Yaskawa INFORM job: A_ROOF_UPPER_0614_2_PAINT_7.JBI

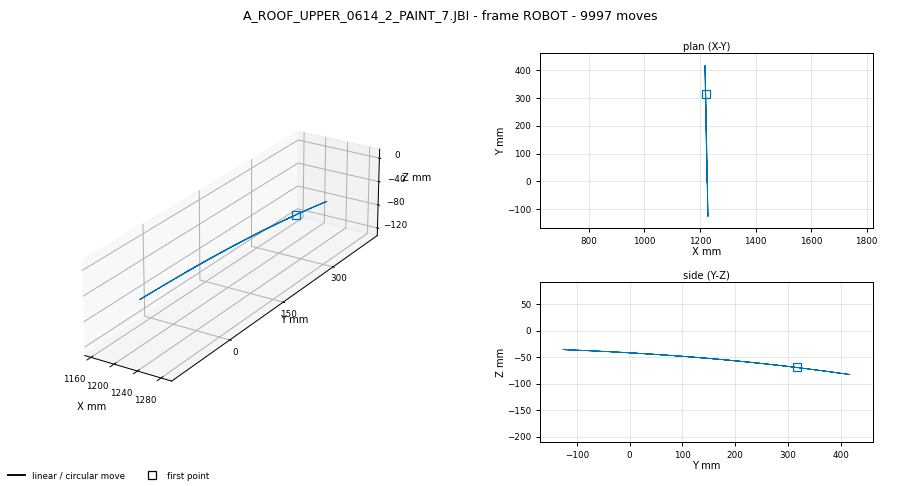
[picture p0: tool path of A_ROOF_UPPER_0614_2_PAINT_7.JBI in frame ROBOT, 9997 of 9997 moves have a stored position in this frame; points joined in program order, loops and branches not executed]
/JOB
//NAME A_ROOF_UPPER_0614_2_PAINT7
//POS
///NPOS 9997,0,0,0,0,0
///TOOL 1
///USER 0
///POSTYPE ROBOT
///RECTAN
///RCONF 1,0,0,0,0,0,0,0,0,0,0,0,0,0,0,0,0,0,0,0,0,0,0,0
C00000=1220.917,316.070,-69.110,-176.284,7.080,148.237
C00001=1220.921,315.822,-69.079,-176.287,7.077,148.237
C00002=1220.925,315.546,-69.046,-176.289,7.074,148.237
C00003=1220.930,315.271,-69.012,-176.291,7.072,148.237
C00004=1220.935,314.994,-68.979,-176.293,7.069,148.237
C00005=1220.939,314.719,-68.945,-176.296,7.066,148.237
C00006=1220.944,314.470,-68.915,-176.298,7.063,148.237
C00007=1220.948,314.222,-68.885,-176.301,7.060,148.237
C00008=1220.953,313.975,-68.854,-176.303,7.058,148.237
C00009=1220.957,313.726,-68.824,-176.306,7.055,148.237
C00010=1220.962,313.478,-68.794,-176.308,7.053,148.237
C00011=1220.966,313.230,-68.764,-176.310,7.051,148.237
C00012=1220.969,312.982,-68.734,-176.312,7.047,148.237
C00013=1220.974,312.733,-68.704,-176.314,7.045,148.237
C00014=1220.978,312.485,-68.673,-176.317,7.042,148.237
C00015=1220.983,312.237,-68.643,-176.319,7.040,148.237
C00016=1220.987,311.989,-68.613,-176.321,7.038,148.237
C00017=1220.991,311.741,-68.582,-176.324,7.035,148.237
C00018=1220.995,311.493,-68.553,-176.326,7.032,148.237
C00019=1221.000,311.245,-68.524,-176.329,7.029,148.237
C00020=1221.004,310.997,-68.493,-176.331,7.027,148.237
C00021=1221.008,310.748,-68.463,-176.333,7.024,148.237
C00022=1221.012,310.501,-68.433,-176.335,7.022,148.237
C00023=1221.017,310.252,-68.403,-176.337,7.019,148.237
C00024=1221.020,310.004,-68.373,-176.340,7.016,148.237
C00025=1221.025,309.755,-68.343,-176.342,7.014,148.237
C00026=1221.030,309.507,-68.313,-176.344,7.011,148.237
C00027=1221.033,309.259,-68.283,-176.347,7.009,148.237
C00028=1221.038,309.011,-68.253,-176.349,7.007,148.237
C00029=1221.042,308.763,-68.223,-176.351,7.004,148.237
C00030=1221.046,308.515,-68.193,-176.353,7.001,148.237
C00031=1221.051,308.266,-68.163,-176.356,6.998,148.237
C00032=1221.055,308.019,-68.133,-176.358,6.996,148.237
C00033=1221.059,307.770,-68.104,-176.360,6.994,148.237
C00034=1221.064,307.522,-68.074,-176.363,6.991,148.237
C00035=1221.068,307.274,-68.043,-176.365,6.989,148.238
C00036=1221.072,307.026,-68.014,-176.367,6.986,148.238
C00037=1221.077,306.778,-67.984,-176.370,6.983,148.238
C00038=1221.081,306.529,-67.955,-176.372,6.981,148.238
C00039=1221.085,306.281,-67.924,-176.375,6.978,148.238
C00040=1221.090,306.033,-67.895,-176.377,6.976,148.238
C00041=1221.094,305.785,-67.865,-176.379,6.974,148.238
C00042=1221.098,305.537,-67.836,-176.382,6.971,148.238
C00043=1221.103,305.288,-67.806,-176.384,6.968,148.238
C00044=1221.107,305.040,-67.776,-176.386,6.965,148.238
C00045=1221.111,304.792,-67.746,-176.388,6.963,148.238
C00046=1221.115,304.544,-67.717,-176.391,6.961,148.238
C00047=1221.119,304.296,-67.687,-176.393,6.958,148.238
C00048=1221.124,304.047,-67.657,-176.395,6.956,148.238
C00049=1221.129,303.799,-67.628,-176.398,6.953,148.238
C00050=1221.133,303.551,-67.599,-176.400,6.950,148.238
C00051=1221.137,303.304,-67.569,-176.402,6.948,148.238
C00052=1221.141,303.055,-67.539,-176.405,6.945,148.238
C00053=1221.145,302.807,-67.510,-176.408,6.943,148.238
C00054=1221.150,302.558,-67.480,-176.410,6.941,148.238
C00055=1221.154,302.310,-67.450,-176.412,6.938,148.238
C00056=1221.159,302.062,-67.421,-176.414,6.936,148.239
C00057=1221.163,301.814,-67.391,-176.417,6.933,148.239
C00058=1221.167,301.565,-67.362,-176.419,6.931,148.239
C00059=1221.171,301.317,-67.332,-176.421,6.928,148.239
C00060=1221.175,301.069,-67.303,-176.424,6.925,148.239
C00061=1221.180,300.821,-67.274,-176.426,6.923,148.239
C00062=1221.184,300.573,-67.244,-176.428,6.921,148.239
C00063=1221.189,300.325,-67.215,-176.431,6.918,148.239
C00064=1221.193,300.076,-67.185,-176.433,6.916,148.239
C00065=1221.198,299.828,-67.155,-176.436,6.913,148.239
C00066=1221.202,299.580,-67.126,-176.438,6.911,148.239
C00067=1221.206,299.331,-67.096,-176.440,6.908,148.239
C00068=1221.210,299.083,-67.067,-176.443,6.905,148.239
C00069=1221.215,298.835,-67.039,-176.445,6.903,148.239
C00070=1221.219,298.587,-67.009,-176.447,6.901,148.239
C00071=1221.224,298.338,-66.980,-176.450,6.898,148.239
C00072=1221.228,298.090,-66.950,-176.453,6.896,148.240
C00073=1221.232,297.842,-66.921,-176.455,6.894,148.240
C00074=1221.236,297.594,-66.891,-176.457,6.891,148.240
C00075=1221.240,297.345,-66.862,-176.459,6.889,148.240
C00076=1221.245,297.097,-66.834,-176.462,6.886,148.240
C00077=1221.249,296.849,-66.805,-176.464,6.883,148.240
C00078=1221.253,296.601,-66.775,-176.467,6.881,148.240
C00079=1221.257,296.353,-66.746,-176.469,6.878,148.240
C00080=1221.261,296.104,-66.716,-176.472,6.876,148.240
C00081=1221.267,295.856,-66.688,-176.474,6.874,148.240
C00082=1221.271,295.608,-66.659,-176.476,6.871,148.240
C00083=1221.275,295.360,-66.629,-176.478,6.869,148.240
C00084=1221.279,295.111,-66.600,-176.481,6.867,148.241
C00085=1221.284,294.862,-66.571,-176.484,6.864,148.241
C00086=1221.288,294.615,-66.542,-176.486,6.862,148.241
C00087=1221.293,294.367,-66.512,-176.488,6.859,148.241
C00088=1221.296,294.118,-66.484,-176.491,6.856,148.241
C00089=1221.300,293.870,-66.455,-176.493,6.854,148.241
C00090=1221.305,293.622,-66.426,-176.495,6.852,148.241
C00091=1221.310,293.373,-66.397,-176.498,6.849,148.241
C00092=1221.314,293.125,-66.367,-176.500,6.847,148.241
C00093=1221.318,292.877,-66.338,-176.503,6.845,148.241
C00094=1221.323,292.629,-66.310,-176.505,6.842,148.241
C00095=1221.327,292.381,-66.281,-176.507,6.840,148.242
C00096=1221.331,292.132,-66.252,-176.510,6.838,148.242
C00097=1221.335,291.884,-66.223,-176.512,6.835,148.242
C00098=1221.340,291.635,-66.194,-176.515,6.833,148.242
C00099=1221.345,291.387,-66.165,-176.517,6.830,148.242
C00100=1221.348,291.138,-66.137,-176.520,6.827,148.242
C00101=1221.352,290.890,-66.107,-176.522,6.825,148.242
C00102=1221.357,290.643,-66.078,-176.524,6.823,148.242
C00103=1221.362,290.394,-66.049,-176.527,6.820,148.242
C00104=1221.365,290.146,-66.020,-176.529,6.818,148.242
C00105=1221.370,289.898,-65.992,-176.532,6.816,148.243
C00106=1221.375,289.623,-65.960,-176.534,6.813,148.243
C00107=1221.380,289.350,-65.928,-176.537,6.810,148.243
C00108=1221.384,289.075,-65.896,-176.540,6.808,148.243
C00109=1221.389,288.801,-65.865,-176.542,6.805,148.243
C00110=1221.394,288.552,-65.836,-176.544,6.803,148.243
C00111=1221.398,288.305,-65.808,-176.548,6.800,148.243
C00112=1221.402,288.056,-65.779,-176.550,6.798,148.243
C00113=1221.406,287.808,-65.749,-176.552,6.796,148.243
C00114=1221.411,287.559,-65.721,-176.555,6.793,148.244
C00115=1221.415,287.311,-65.693,-176.557,6.791,148.244
C00116=1221.419,287.062,-65.663,-176.559,6.789,148.244
C00117=1221.424,286.814,-65.635,-176.562,6.787,148.244
C00118=1221.428,286.566,-65.607,-176.564,6.784,148.244
C00119=1221.433,286.318,-65.578,-176.567,6.781,148.244
C00120=1221.437,286.070,-65.550,-176.569,6.780,148.244
C00121=1221.441,285.821,-65.521,-176.572,6.776,148.244
C00122=1221.446,285.573,-65.493,-176.574,6.774,148.245
C00123=1221.450,285.325,-65.464,-176.577,6.772,148.245
C00124=1221.455,285.076,-65.435,-176.579,6.769,148.245
C00125=1221.459,284.828,-65.407,-176.581,6.767,148.245
C00126=1221.463,284.579,-65.378,-176.584,6.765,148.245
C00127=1221.468,284.331,-65.349,-176.586,6.763,148.245
C00128=1221.472,284.083,-65.321,-176.589,6.760,148.245
C00129=1221.477,283.835,-65.293,-176.591,6.758,148.246
C00130=1221.480,283.586,-65.265,-176.593,6.756,148.246
C00131=1221.485,283.337,-65.236,-176.596,6.753,148.246
C00132=1221.489,283.090,-65.207,-176.599,6.751,148.246
C00133=1221.494,282.841,-65.179,-176.601,6.749,148.246
C00134=1221.499,282.593,-65.150,-176.603,6.747,148.246
C00135=1221.502,282.344,-65.122,-176.606,6.744,148.246
C00136=1221.507,282.096,-65.094,-176.608,6.742,148.246
C00137=1221.511,281.847,-65.066,-176.610,6.739,148.246
C00138=1221.516,281.599,-65.037,-176.614,6.737,148.247
C00139=1221.520,281.351,-65.009,-176.616,6.734,148.247
C00140=1221.524,281.103,-64.981,-176.618,6.733,148.247
C00141=1221.529,280.854,-64.953,-176.620,6.730,148.247
C00142=1221.533,280.605,-64.925,-176.623,6.727,148.247
C00143=1221.537,280.358,-64.895,-176.626,6.725,148.247
C00144=1221.541,280.109,-64.867,-176.628,6.723,148.248
C00145=1221.546,279.861,-64.839,-176.630,6.721,148.248
C00146=1221.550,279.612,-64.811,-176.633,6.718,148.248
C00147=1221.555,279.364,-64.782,-176.635,6.716,148.248
C00148=1221.559,279.115,-64.755,-176.638,6.714,148.248
C00149=1221.563,278.867,-64.727,-176.640,6.711,148.248
C00150=1221.568,278.618,-64.698,-176.643,6.709,148.249
C00151=1221.572,278.370,-64.671,-176.645,6.707,148.249
C00152=1221.577,278.122,-64.642,-176.647,6.705,148.249
C00153=1221.581,277.874,-64.614,-176.650,6.702,148.249
C00154=1221.585,277.625,-64.586,-176.653,6.700,148.249
C00155=1221.590,277.377,-64.558,-176.655,6.698,148.249
C00156=1221.594,277.129,-64.530,-176.657,6.696,148.249
C00157=1221.598,276.880,-64.502,-176.660,6.693,148.250
C00158=1221.603,276.632,-64.473,-176.663,6.691,148.250
C00159=1221.607,276.383,-64.446,-176.665,6.689,148.250
C00160=1221.612,276.135,-64.418,-176.667,6.687,148.250
C00161=1221.616,275.886,-64.389,-176.670,6.684,148.250
C00162=1221.620,275.638,-64.362,-176.673,6.682,148.250
C00163=1221.624,275.390,-64.334,-176.675,6.680,148.250
C00164=1221.629,275.142,-64.305,-176.677,6.678,148.251
C00165=1221.634,274.893,-64.278,-176.679,6.676,148.251
C00166=1221.638,274.645,-64.250,-176.683,6.673,148.251
C00167=1221.642,274.397,-64.222,-176.685,6.671,148.251
C00168=1221.647,274.148,-64.193,-176.687,6.669,148.251
C00169=1221.651,273.899,-64.166,-176.689,6.667,148.251
C00170=1221.656,273.651,-64.139,-176.693,6.664,148.252
C00171=1221.659,273.403,-64.110,-176.695,6.662,148.252
C00172=1221.665,273.154,-64.083,-176.697,6.660,148.252
C00173=1221.668,272.905,-64.055,-176.699,6.658,148.252
C00174=1221.673,272.658,-64.027,-176.703,6.655,148.252
C00175=1221.677,272.409,-64.000,-176.705,6.653,148.253
C00176=1221.682,272.160,-63.971,-176.707,6.650,148.253
C00177=1221.686,271.912,-63.943,-176.709,6.649,148.253
C00178=1221.691,271.664,-63.916,-176.712,6.646,148.253
C00179=1221.695,271.415,-63.888,-176.715,6.644,148.253
C00180=1221.699,271.167,-63.860,-176.717,6.641,148.253
C00181=1221.704,270.919,-63.833,-176.719,6.640,148.254
C00182=1221.708,270.670,-63.805,-176.722,6.637,148.254
C00183=1221.713,270.422,-63.777,-176.724,6.635,148.254
C00184=1221.717,270.174,-63.750,-176.727,6.633,148.254
C00185=1221.721,269.924,-63.722,-176.729,6.631,148.254
C00186=1221.726,269.677,-63.694,-176.732,6.629,148.255
C00187=1221.730,269.429,-63.667,-176.734,6.626,148.255
C00188=1221.734,269.180,-63.639,-176.737,6.624,148.255
C00189=1221.739,268.931,-63.611,-176.739,6.622,148.255
C00190=1221.744,268.683,-63.584,-176.742,6.620,148.255
C00191=1221.747,268.434,-63.556,-176.744,6.617,148.255
C00192=1221.752,268.186,-63.529,-176.747,6.616,148.256
C00193=1221.757,267.937,-63.502,-176.749,6.613,148.256
C00194=1221.761,267.689,-63.473,-176.752,6.611,148.256
C00195=1221.765,267.440,-63.446,-176.754,6.608,148.256
C00196=1221.770,267.192,-63.419,-176.757,6.607,148.256
C00197=1221.774,266.944,-63.392,-176.759,6.604,148.256
C00198=1221.778,266.695,-63.363,-176.762,6.602,148.257
C00199=1221.783,266.447,-63.336,-176.764,6.599,148.257
C00200=1221.787,266.198,-63.309,-176.767,6.598,148.257
C00201=1221.792,265.950,-63.282,-176.769,6.596,148.257
C00202=1221.796,265.701,-63.254,-176.772,6.593,148.257
C00203=1221.800,265.453,-63.227,-176.774,6.592,148.258
C00204=1221.805,265.205,-63.199,-176.777,6.589,148.258
C00205=1221.809,264.956,-63.172,-176.779,6.587,148.258
C00206=1221.813,264.707,-63.145,-176.782,6.584,148.258
C00207=1221.818,264.459,-63.117,-176.784,6.583,148.258
C00208=1221.822,264.211,-63.090,-176.787,6.581,148.259
C00209=1221.827,263.962,-63.063,-176.789,6.579,148.259
C00210=1221.832,263.690,-63.033,-176.792,6.576,148.259
C00211=1221.836,263.417,-63.002,-176.795,6.574,148.259
C00212=1221.842,263.144,-62.972,-176.797,6.571,148.259
C00213=1221.846,262.872,-62.942,-176.800,6.569,148.260
C00214=1221.851,262.623,-62.915,-176.803,6.567,148.260
C00215=1221.855,262.375,-62.888,-176.805,6.564,148.260
C00216=1221.860,262.126,-62.861,-176.808,6.562,148.260
C00217=1221.864,261.877,-62.834,-176.810,6.560,148.260
C00218=1221.868,261.629,-62.806,-176.813,6.558,148.261
C00219=1221.873,261.381,-62.779,-176.815,6.556,148.261
C00220=1221.877,261.132,-62.753,-176.817,6.554,148.261
C00221=1221.882,260.884,-62.725,-176.820,6.551,148.261
C00222=1221.886,260.635,-62.698,-176.823,6.549,148.261
C00223=1221.890,260.386,-62.671,-176.825,6.547,148.262
C00224=1221.895,260.138,-62.644,-176.828,6.545,148.262
C00225=1221.900,259.889,-62.617,-176.830,6.543,148.262
C00226=1221.904,259.641,-62.590,-176.833,6.541,148.262
C00227=1221.908,259.393,-62.563,-176.835,6.539,148.263
C00228=1221.913,259.145,-62.536,-176.838,6.536,148.263
C00229=1221.917,258.896,-62.508,-176.840,6.534,148.263
C00230=1221.922,258.648,-62.481,-176.843,6.532,148.263
C00231=1221.926,258.399,-62.454,-176.845,6.530,148.263
C00232=1221.930,258.150,-62.428,-176.848,6.529,148.264
C00233=1221.935,257.902,-62.400,-176.850,6.526,148.264
C00234=1221.939,257.653,-62.373,-176.853,6.524,148.264
C00235=1221.944,257.405,-62.346,-176.855,6.523,148.264
C00236=1221.948,257.157,-62.320,-176.858,6.520,148.265
C00237=1221.952,256.908,-62.293,-176.860,6.518,148.265
C00238=1221.957,256.660,-62.266,-176.863,6.516,148.265
C00239=1221.962,256.411,-62.239,-176.865,6.514,148.265
C00240=1221.966,256.162,-62.213,-176.868,6.512,148.266
C00241=1221.970,255.913,-62.185,-176.870,6.510,148.266
C00242=1221.975,255.665,-62.158,-176.873,6.508,148.266
C00243=1221.979,255.416,-62.132,-176.875,6.506,148.266
C00244=1221.983,255.168,-62.105,-176.878,6.503,148.266
C00245=1221.988,254.920,-62.078,-176.880,6.501,148.267
C00246=1221.993,254.671,-62.051,-176.883,6.499,148.267
C00247=1221.996,254.423,-62.024,-176.885,6.497,148.267
C00248=1222.001,254.174,-61.998,-176.888,6.495,148.267
C00249=1222.006,253.925,-61.971,-176.890,6.493,148.268
C00250=1222.010,253.677,-61.944,-176.893,6.491,148.268
C00251=1222.015,253.429,-61.917,-176.895,6.489,148.268
C00252=1222.019,253.180,-61.891,-176.898,6.487,148.268
C00253=1222.024,252.931,-61.865,-176.900,6.484,148.268
C00254=1222.028,252.683,-61.838,-176.903,6.482,148.269
C00255=1222.032,252.435,-61.811,-176.906,6.480,148.269
C00256=1222.037,252.186,-61.784,-176.908,6.478,148.269
C00257=1222.042,251.937,-61.758,-176.910,6.476,148.269
C00258=1222.046,251.689,-61.731,-176.913,6.474,148.270
C00259=1222.050,251.440,-61.704,-176.916,6.472,148.270
C00260=1222.055,251.191,-61.678,-176.918,6.470,148.270
C00261=1222.059,250.943,-61.651,-176.920,6.468,148.270
C00262=1222.063,250.695,-61.625,-176.923,6.467,148.271
C00263=1222.068,250.446,-61.598,-176.925,6.464,148.271
C00264=1222.073,250.197,-61.571,-176.928,6.462,148.271
C00265=1222.077,249.949,-61.545,-176.931,6.460,148.271
C00266=1222.082,249.700,-61.519,-176.934,6.458,148.272
C00267=1222.086,249.452,-61.492,-176.936,6.456,148.272
C00268=1222.090,249.203,-61.465,-176.938,6.454,148.272
C00269=1222.094,248.954,-61.439,-176.941,6.452,148.272
C00270=1222.099,248.706,-61.412,-176.943,6.450,148.272
C00271=1222.103,248.457,-61.387,-176.946,6.448,148.273
C00272=1222.108,248.209,-61.359,-176.948,6.446,148.273
C00273=1222.113,247.960,-61.334,-176.951,6.444,148.273
C00274=1222.117,247.712,-61.307,-176.953,6.442,148.273
C00275=1222.121,247.464,-61.281,-176.956,6.440,148.274
C00276=1222.126,247.215,-61.254,-176.958,6.438,148.274
C00277=1222.130,246.967,-61.228,-176.960,6.436,148.274
C00278=1222.134,246.718,-61.202,-176.963,6.434,148.274
C00279=1222.139,246.469,-61.175,-176.966,6.431,148.275
C00280=1222.143,246.220,-61.149,-176.969,6.430,148.275
C00281=1222.148,245.971,-61.123,-176.971,6.427,148.275
C00282=1222.152,245.723,-61.096,-176.974,6.425,148.275
C00283=1222.158,245.475,-61.070,-176.976,6.424,148.276
C00284=1222.162,245.227,-61.044,-176.979,6.422,148.276
C00285=1222.166,244.978,-61.018,-176.981,6.419,148.276
C00286=1222.171,244.729,-60.991,-176.984,6.418,148.276
C00287=1222.175,244.480,-60.965,-176.986,6.416,148.277
C00288=1222.180,244.231,-60.939,-176.989,6.414,148.277
C00289=1222.184,243.983,-60.913,-176.991,6.412,148.277
C00290=1222.188,243.734,-60.887,-176.994,6.410,148.277
C00291=1222.194,243.486,-60.861,-176.996,6.408,148.278
C00292=1222.197,243.238,-60.834,-176.999,6.406,148.278
C00293=1222.202,242.989,-60.809,-177.001,6.404,148.278
C00294=1222.207,242.740,-60.782,-177.004,6.402,148.279
C00295=1222.211,242.492,-60.756,-177.006,6.400,148.279
C00296=1222.215,242.243,-60.730,-177.009,6.398,148.279
C00297=1222.220,241.994,-60.704,-177.011,6.396,148.279
C00298=1222.224,241.746,-60.678,-177.013,6.394,148.280
C00299=1222.228,241.497,-60.652,-177.016,6.392,148.280
C00300=1222.233,241.249,-60.626,-177.019,6.390,148.280
C00301=1222.238,240.999,-60.600,-177.022,6.388,148.280
C00302=1222.242,240.752,-60.574,-177.024,6.386,148.281
C00303=1222.246,240.503,-60.548,-177.027,6.384,148.281
C00304=1222.251,240.254,-60.522,-177.029,6.382,148.281
C00305=1222.256,240.005,-60.496,-177.032,6.380,148.281
C00306=1222.260,239.756,-60.470,-177.035,6.378,148.282
C00307=1222.264,239.509,-60.444,-177.037,6.376,148.282
C00308=1222.269,239.260,-60.418,-177.039,6.374,148.282
C00309=1222.274,239.011,-60.392,-177.042,6.372,148.283
C00310=1222.278,238.762,-60.366,-177.045,6.370,148.283
C00311=1222.283,238.514,-60.341,-177.047,6.368,148.283
C00312=1222.287,238.265,-60.315,-177.049,6.366,148.283
C00313=1222.291,238.017,-60.289,-177.052,6.364,148.284
C00314=1222.296,237.745,-60.260,-177.055,6.363,148.284
C00315=1222.301,237.474,-60.232,-177.057,6.361,148.284
C00316=1222.306,237.202,-60.204,-177.060,6.358,148.284
C00317=1222.311,236.931,-60.176,-177.063,6.356,148.285
C00318=1222.315,236.682,-60.150,-177.066,6.354,148.285
C00319=1222.320,236.434,-60.124,-177.068,6.352,148.285
C00320=1222.324,236.186,-60.099,-177.070,6.350,148.286
C00321=1222.329,235.937,-60.073,-177.073,6.348,148.286
C00322=1222.333,235.688,-60.047,-177.076,6.346,148.286
C00323=1222.338,235.439,-60.021,-177.078,6.345,148.286
C00324=1222.343,235.191,-59.996,-177.081,6.343,148.287
C00325=1222.347,234.942,-59.970,-177.083,6.341,148.287
C00326=1222.351,234.693,-59.944,-177.086,6.339,148.287
C00327=1222.356,234.445,-59.919,-177.088,6.337,148.288
C00328=1222.360,234.196,-59.893,-177.091,6.335,148.288
C00329=1222.364,233.947,-59.867,-177.093,6.333,148.288
C00330=1222.369,233.699,-59.842,-177.096,6.331,148.288
C00331=1222.374,233.450,-59.817,-177.099,6.329,148.289
C00332=1222.378,233.201,-59.791,-177.101,6.327,148.289
C00333=1222.383,232.953,-59.766,-177.103,6.325,148.289
C00334=1222.387,232.704,-59.740,-177.106,6.323,148.290
C00335=1222.391,232.455,-59.714,-177.109,6.321,148.290
C00336=1222.396,232.207,-59.689,-177.111,6.320,148.290
C00337=1222.400,231.958,-59.663,-177.114,6.318,148.291
C00338=1222.404,231.710,-59.637,-177.117,6.316,148.291
C00339=1222.410,231.461,-59.613,-177.119,6.314,148.291
C00340=1222.414,231.212,-59.587,-177.121,6.312,148.291
C00341=1222.419,230.964,-59.561,-177.124,6.310,148.292
C00342=1222.423,230.715,-59.536,-177.127,6.308,148.292
C00343=1222.427,230.466,-59.511,-177.129,6.306,148.292
C00344=1222.432,230.218,-59.485,-177.132,6.304,148.293
C00345=1222.436,229.969,-59.460,-177.134,6.303,148.293
C00346=1222.441,229.721,-59.434,-177.136,6.301,148.293
C00347=1222.446,229.471,-59.409,-177.139,6.299,148.293
C00348=1222.450,229.223,-59.383,-177.141,6.297,148.294
C00349=1222.455,228.974,-59.358,-177.144,6.296,148.294
C00350=1222.459,228.726,-59.332,-177.147,6.294,148.294
C00351=1222.464,228.477,-59.308,-177.149,6.292,148.295
C00352=1222.468,228.228,-59.282,-177.152,6.290,148.295
C00353=1222.473,227.979,-59.256,-177.154,6.288,148.295
C00354=1222.477,227.731,-59.232,-177.157,6.286,148.296
C00355=1222.481,227.482,-59.206,-177.159,6.284,148.296
C00356=1222.486,227.234,-59.181,-177.162,6.282,148.296
C00357=1222.491,226.985,-59.156,-177.164,6.280,148.296
C00358=1222.495,226.736,-59.130,-177.167,6.278,148.297
C00359=1222.500,226.487,-59.105,-177.170,6.277,148.297
C00360=1222.505,226.239,-59.080,-177.172,6.275,148.297
C00361=1222.508,225.990,-59.055,-177.175,6.273,148.298
C00362=1222.513,225.742,-59.030,-177.178,6.271,148.298
C00363=1222.518,225.493,-59.004,-177.180,6.269,148.298
C00364=1222.522,225.243,-58.979,-177.183,6.267,148.299
C00365=1222.527,224.995,-58.954,-177.185,6.265,148.299
C00366=1222.532,224.746,-58.929,-177.188,6.263,148.299
C00367=1222.536,224.498,-58.904,-177.190,6.262,148.299
C00368=1222.540,224.249,-58.879,-177.192,6.260,148.300
C00369=1222.545,224.001,-58.854,-177.195,6.259,148.300
C00370=1222.550,223.751,-58.829,-177.198,6.257,148.300
C00371=1222.554,223.503,-58.804,-177.200,6.255,148.301
C00372=1222.559,223.255,-58.779,-177.203,6.253,148.301
C00373=1222.563,223.006,-58.754,-177.205,6.251,148.301
C00374=1222.568,222.757,-58.729,-177.208,6.249,148.302
C00375=1222.572,222.509,-58.704,-177.211,6.247,148.302
C00376=1222.577,222.260,-58.679,-177.213,6.246,148.302
C00377=1222.581,222.011,-58.654,-177.216,6.244,148.303
C00378=1222.586,221.762,-58.629,-177.218,6.241,148.303
C00379=1222.590,221.513,-58.604,-177.221,6.240,148.303
C00380=1222.595,221.265,-58.580,-177.223,6.238,148.303
C00381=1222.599,221.016,-58.554,-177.226,6.236,148.304
C00382=1222.604,220.767,-58.530,-177.229,6.234,148.304
C00383=1222.608,220.519,-58.504,-177.231,6.233,148.304
C00384=1222.613,220.270,-58.479,-177.233,6.231,148.305
C00385=1222.617,220.021,-58.455,-177.236,6.229,148.305
C00386=1222.622,219.773,-58.429,-177.239,6.227,148.305
C00387=1222.627,219.524,-58.405,-177.241,6.226,148.306
C00388=1222.631,219.275,-58.380,-177.244,6.224,148.306
C00389=1222.636,219.026,-58.356,-177.246,6.222,148.306
C00390=1222.640,218.777,-58.330,-177.249,6.220,148.307
C00391=1222.644,218.529,-58.306,-177.252,6.218,148.307
C00392=1222.649,218.280,-58.281,-177.254,6.216,148.307
C00393=1222.653,218.031,-58.257,-177.257,6.214,148.308
C00394=1222.658,217.783,-58.231,-177.260,6.213,148.308
C00395=1222.663,217.534,-58.207,-177.262,6.212,148.308
C00396=1222.667,217.285,-58.182,-177.264,6.210,148.309
C00397=1222.672,217.036,-58.158,-177.267,6.208,148.309
C00398=1222.676,216.787,-58.133,-177.270,6.206,148.309
C00399=1222.681,216.539,-58.108,-177.272,6.204,148.310
C00400=1222.685,216.291,-58.084,-177.275,6.202,148.310
C00401=1222.690,216.041,-58.059,-177.277,6.200,148.310
C00402=1222.694,215.793,-58.035,-177.280,6.199,148.311
C00403=1222.699,215.544,-58.010,-177.283,6.197,148.311
C00404=1222.704,215.295,-57.985,-177.285,6.195,148.311
C00405=1222.708,215.046,-57.961,-177.288,6.193,148.312
C00406=1222.713,214.798,-57.936,-177.291,6.191,148.312
C00407=1222.717,214.548,-57.912,-177.293,6.190,148.312
C00408=1222.722,214.300,-57.886,-177.295,6.188,148.313
C00409=1222.726,214.052,-57.862,-177.298,6.186,148.313
C00410=1222.731,213.803,-57.837,-177.301,6.185,148.313
C00411=1222.735,213.554,-57.813,-177.303,6.183,148.314
C00412=1222.740,213.306,-57.789,-177.306,6.181,148.314
C00413=1222.744,213.056,-57.764,-177.308,6.179,148.314
C00414=1222.748,212.808,-57.740,-177.311,6.177,148.315
C00415=1222.754,212.559,-57.715,-177.314,6.175,148.315
C00416=1222.758,212.311,-57.691,-177.316,6.174,148.315
C00417=1222.763,212.061,-57.666,-177.318,6.172,148.316
C00418=1222.768,211.791,-57.640,-177.321,6.171,148.316
C00419=1222.772,211.521,-57.614,-177.324,6.168,148.316
C00420=1222.778,211.250,-57.587,-177.327,6.166,148.317
C00421=1222.782,210.980,-57.560,-177.330,6.164,148.317
C00422=1222.787,210.731,-57.536,-177.332,6.162,148.317
C00423=1222.792,210.482,-57.512,-177.335,6.160,148.318
C00424=1222.796,210.233,-57.488,-177.337,6.159,148.318
C00425=1222.800,209.984,-57.464,-177.340,6.158,148.318
C00426=1222.805,209.736,-57.439,-177.342,6.156,148.319
C00427=1222.810,209.487,-57.415,-177.345,6.154,148.319
C00428=1222.815,209.238,-57.390,-177.347,6.152,148.319
C00429=1222.819,208.989,-57.366,-177.350,6.150,148.320
C00430=1222.823,208.741,-57.342,-177.353,6.149,148.320
C00431=1222.828,208.492,-57.318,-177.356,6.147,148.321
C00432=1222.833,208.243,-57.294,-177.358,6.146,148.321
C00433=1222.837,207.995,-57.270,-177.361,6.144,148.321
C00434=1222.842,207.745,-57.245,-177.363,6.142,148.322
C00435=1222.846,207.496,-57.221,-177.366,6.140,148.322
C00436=1222.851,207.248,-57.197,-177.368,6.138,148.322
C00437=1222.855,206.999,-57.173,-177.371,6.137,148.323
C00438=1222.860,206.751,-57.148,-177.373,6.136,148.323
C00439=1222.864,206.501,-57.125,-177.376,6.134,148.323
C00440=1222.869,206.253,-57.101,-177.378,6.132,148.324
C00441=1222.874,206.004,-57.076,-177.381,6.130,148.324
C00442=1222.878,205.755,-57.052,-177.384,6.128,148.324
C00443=1222.883,205.506,-57.029,-177.386,6.126,148.325
C00444=1222.887,205.258,-57.004,-177.389,6.124,148.325
C00445=1222.891,205.009,-56.980,-177.391,6.123,148.326
C00446=1222.897,204.760,-56.956,-177.394,6.122,148.326
C00447=1222.901,204.511,-56.932,-177.396,6.120,148.326
C00448=1222.905,204.263,-56.908,-177.399,6.118,148.327
C00449=1222.910,204.014,-56.885,-177.402,6.116,148.327
C00450=1222.915,203.765,-56.860,-177.404,6.114,148.327
C00451=1222.920,203.516,-56.837,-177.407,6.113,148.328
C00452=1222.924,203.267,-56.812,-177.409,6.112,148.328
C00453=1222.928,203.018,-56.788,-177.412,6.110,148.328
C00454=1222.933,202.769,-56.765,-177.415,6.108,148.329
C00455=1222.937,202.521,-56.741,-177.417,6.106,148.329
C00456=1222.943,202.272,-56.717,-177.419,6.105,148.330
C00457=1222.947,202.023,-56.693,-177.422,6.103,148.330
C00458=1222.952,201.774,-56.669,-177.425,6.101,148.330
C00459=1222.956,201.526,-56.645,-177.427,6.100,148.331
C00460=1222.960,201.276,-56.621,-177.430,6.098,148.331
C00461=1222.965,201.028,-56.597,-177.433,6.096,148.331
C00462=1222.969,200.779,-56.574,-177.435,6.095,148.332
C00463=1222.974,200.530,-56.550,-177.437,6.093,148.332
C00464=1222.979,200.281,-56.527,-177.440,6.091,148.332
C00465=1222.984,200.032,-56.502,-177.443,6.090,148.333
C00466=1222.988,199.783,-56.479,-177.446,6.088,148.333
C00467=1222.993,199.535,-56.454,-177.448,6.087,148.334
C00468=1222.997,199.286,-56.431,-177.451,6.085,148.334
C00469=1223.002,199.038,-56.407,-177.453,6.083,148.334
C00470=1223.007,198.789,-56.384,-177.456,6.081,148.335
C00471=1223.011,198.539,-56.360,-177.458,6.079,148.335
C00472=1223.016,198.291,-56.336,-177.461,6.078,148.335
C00473=1223.020,198.042,-56.313,-177.463,6.077,148.336
C00474=1223.025,197.793,-56.290,-177.466,6.075,148.336
C00475=1223.029,197.545,-56.265,-177.469,6.073,148.337
C00476=1223.034,197.296,-56.242,-177.471,6.072,148.337
C00477=1223.039,197.047,-56.219,-177.474,6.070,148.337
C00478=1223.043,196.798,-56.195,-177.476,6.068,148.338
C00479=1223.048,196.549,-56.171,-177.479,6.067,148.338
C00480=1223.053,196.300,-56.148,-177.482,6.065,148.338
C00481=1223.057,196.052,-56.124,-177.484,6.064,148.339
C00482=1223.062,195.803,-56.100,-177.486,6.062,148.339
C00483=1223.066,195.554,-56.077,-177.489,6.060,148.339
C00484=1223.071,195.305,-56.054,-177.492,6.058,148.340
C00485=1223.075,195.056,-56.030,-177.494,6.058,148.340
C00486=1223.080,194.807,-56.006,-177.497,6.056,148.341
C00487=1223.085,194.558,-55.983,-177.499,6.054,148.341
C00488=1223.090,194.309,-55.960,-177.502,6.052,148.341
C00489=1223.094,194.061,-55.936,-177.505,6.050,148.342
C00490=1223.098,193.812,-55.913,-177.507,6.049,148.342
C00491=1223.103,193.563,-55.889,-177.509,6.047,148.342
C00492=1223.107,193.314,-55.866,-177.512,6.045,148.343
C00493=1223.112,193.065,-55.843,-177.515,6.044,148.343
C00494=1223.117,192.816,-55.819,-177.517,6.043,148.344
C00495=1223.121,192.567,-55.795,-177.520,6.041,148.344
C00496=1223.126,192.318,-55.772,-177.523,6.039,148.344
C00497=1223.131,192.069,-55.749,-177.525,6.037,148.345
C00498=1223.135,191.820,-55.725,-177.527,6.036,148.345
C00499=1223.139,191.572,-55.702,-177.530,6.035,148.345
C00500=1223.144,191.323,-55.679,-177.533,6.033,148.346
C00501=1223.149,191.074,-55.656,-177.536,6.031,148.346
C00502=1223.154,190.825,-55.633,-177.538,6.030,148.347
C00503=1223.159,190.576,-55.609,-177.540,6.028,148.347
C00504=1223.163,190.327,-55.586,-177.543,6.027,148.347
C00505=1223.167,190.078,-55.563,-177.546,6.025,148.348
C00506=1223.172,189.829,-55.540,-177.548,6.024,148.348
C00507=1223.177,189.580,-55.517,-177.551,6.022,148.349
C00508=1223.181,189.331,-55.493,-177.554,6.020,148.349
C00509=1223.186,189.082,-55.470,-177.556,6.019,148.350
C00510=1223.191,188.834,-55.447,-177.558,6.018,148.350
C00511=1223.195,188.585,-55.424,-177.561,6.016,148.350
C00512=1223.200,188.336,-55.401,-177.564,6.014,148.351
C00513=1223.205,188.087,-55.377,-177.566,6.013,148.351
C00514=1223.209,187.838,-55.355,-177.569,6.011,148.352
C00515=1223.213,187.589,-55.331,-177.572,6.009,148.352
C00516=1223.218,187.340,-55.308,-177.574,6.008,148.352
C00517=1223.222,187.092,-55.285,-177.576,6.007,148.353
C00518=1223.227,186.843,-55.262,-177.579,6.005,148.353
C00519=1223.232,186.594,-55.239,-177.582,6.003,148.353
C00520=1223.237,186.345,-55.215,-177.584,6.002,148.354
C00521=1223.241,186.097,-55.193,-177.587,6.000,148.354
C00522=1223.246,185.827,-55.168,-177.589,5.999,148.355
C00523=1223.251,185.557,-55.143,-177.593,5.997,148.355
C00524=1223.256,185.288,-55.118,-177.595,5.995,148.356
C00525=1223.261,185.018,-55.093,-177.598,5.993,148.356
C00526=1223.266,184.769,-55.070,-177.601,5.992,148.356
C00527=1223.270,184.520,-55.047,-177.603,5.991,148.357
C00528=1223.276,184.271,-55.025,-177.606,5.989,148.357
C00529=1223.279,184.022,-55.002,-177.608,5.987,148.358
C00530=1223.284,183.773,-54.979,-177.610,5.986,148.358
C00531=1223.289,183.524,-54.955,-177.613,5.984,148.358
C00532=1223.293,183.275,-54.933,-177.616,5.983,148.359
C00533=1223.298,183.027,-54.910,-177.618,5.982,148.359
C00534=1223.303,182.778,-54.887,-177.621,5.980,148.360
C00535=1223.307,182.529,-54.864,-177.624,5.978,148.360
C00536=1223.312,182.279,-54.841,-177.626,5.976,148.360
C00537=1223.317,182.031,-54.819,-177.629,5.976,148.361
C00538=1223.321,181.782,-54.796,-177.632,5.974,148.361
C00539=1223.326,181.533,-54.774,-177.634,5.972,148.362
C00540=1223.330,181.284,-54.750,-177.636,5.971,148.362
C00541=1223.336,181.035,-54.727,-177.639,5.969,148.362
C00542=1223.340,180.786,-54.705,-177.642,5.968,148.363
C00543=1223.345,180.537,-54.682,-177.644,5.967,148.363
C00544=1223.349,180.288,-54.659,-177.647,5.965,148.364
C00545=1223.354,180.039,-54.637,-177.649,5.963,148.364
C00546=1223.358,179.791,-54.614,-177.652,5.962,148.364
C00547=1223.363,179.542,-54.591,-177.655,5.961,148.365
C00548=1223.368,179.293,-54.569,-177.657,5.959,148.365
C00549=1223.372,179.044,-54.546,-177.659,5.958,148.366
C00550=1223.377,178.795,-54.524,-177.662,5.956,148.366
C00551=1223.381,178.546,-54.500,-177.665,5.954,148.366
C00552=1223.386,178.297,-54.479,-177.667,5.953,148.367
C00553=1223.391,178.048,-54.455,-177.670,5.952,148.367
C00554=1223.395,177.799,-54.433,-177.673,5.950,148.368
C00555=1223.401,177.550,-54.410,-177.675,5.949,148.368
C00556=1223.405,177.301,-54.388,-177.678,5.947,148.369
C00557=1223.409,177.052,-54.365,-177.681,5.945,148.369
C00558=1223.414,176.803,-54.343,-177.683,5.944,148.369
C00559=1223.418,176.555,-54.320,-177.685,5.943,148.370
C00560=1223.423,176.305,-54.298,-177.688,5.941,148.370
C00561=1223.428,176.057,-54.275,-177.690,5.940,148.371
C00562=1223.433,175.807,-54.253,-177.693,5.938,148.371
C00563=1223.437,175.558,-54.230,-177.695,5.937,148.371
C00564=1223.442,175.310,-54.208,-177.698,5.935,148.372
C00565=1223.446,175.061,-54.185,-177.701,5.934,148.372
C00566=1223.451,174.812,-54.163,-177.703,5.933,148.373
C00567=1223.456,174.563,-54.141,-177.706,5.931,148.373
C00568=1223.460,174.314,-54.118,-177.708,5.929,148.374
C00569=1223.465,174.065,-54.096,-177.711,5.929,148.374
C00570=1223.470,173.816,-54.073,-177.714,5.927,148.375
C00571=1223.474,173.567,-54.051,-177.716,5.925,148.375
C00572=1223.479,173.318,-54.029,-177.718,5.924,148.375
C00573=1223.484,173.069,-54.006,-177.722,5.922,148.376
C00574=1223.489,172.820,-53.984,-177.724,5.921,148.376
C00575=1223.493,172.571,-53.962,-177.726,5.920,148.377
C00576=1223.498,172.322,-53.938,-177.729,5.918,148.377
C00577=1223.502,172.073,-53.917,-177.732,5.917,148.378
C00578=1223.507,171.824,-53.895,-177.734,5.915,148.378
C00579=1223.512,171.575,-53.873,-177.737,5.913,148.378
C00580=1223.516,171.326,-53.850,-177.739,5.912,148.379
C00581=1223.521,171.078,-53.828,-177.742,5.911,148.379
C00582=1223.525,170.828,-53.806,-177.744,5.910,148.380
C00583=1223.530,170.579,-53.783,-177.747,5.908,148.380
C00584=1223.535,170.331,-53.761,-177.750,5.906,148.380
C00585=1223.539,170.081,-53.739,-177.752,5.906,148.381
C00586=1223.544,169.833,-53.717,-177.755,5.904,148.381
C00587=1223.549,169.583,-53.695,-177.757,5.903,148.382
C00588=1223.554,169.334,-53.673,-177.760,5.901,148.382
C00589=1223.558,169.086,-53.650,-177.763,5.899,148.383
C00590=1223.563,168.837,-53.628,-177.765,5.898,148.383
C00591=1223.568,168.587,-53.606,-177.767,5.897,148.383
C00592=1223.573,168.339,-53.584,-177.770,5.896,148.384
C00593=1223.577,168.089,-53.562,-177.773,5.894,148.384
C00594=1223.582,167.841,-53.540,-177.775,5.892,148.385
C00595=1223.586,167.592,-53.518,-177.778,5.892,148.385
C00596=1223.591,167.344,-53.496,-177.781,5.890,148.386
C00597=1223.596,167.094,-53.473,-177.783,5.889,148.386
C00598=1223.600,166.845,-53.452,-177.785,5.887,148.386
C00599=1223.605,166.596,-53.430,-177.788,5.886,148.387
C00600=1223.610,166.347,-53.408,-177.791,5.885,148.387
C00601=1223.614,166.098,-53.386,-177.793,5.883,148.388
C00602=1223.619,165.849,-53.364,-177.796,5.882,148.388
C00603=1223.623,165.600,-53.342,-177.798,5.880,148.389
C00604=1223.629,165.351,-53.320,-177.801,5.878,148.389
C00605=1223.633,165.102,-53.298,-177.804,5.878,148.390
C00606=1223.638,164.853,-53.276,-177.806,5.876,148.390
C00607=1223.642,164.604,-53.254,-177.808,5.875,148.391
C00608=1223.647,164.355,-53.232,-177.811,5.873,148.391
C00609=1223.651,164.106,-53.210,-177.814,5.872,148.392
C00610=1223.656,163.857,-53.189,-177.816,5.871,148.392
C00611=1223.661,163.608,-53.167,-177.819,5.869,148.392
C00612=1223.665,163.359,-53.145,-177.822,5.868,148.393
C00613=1223.670,163.110,-53.123,-177.824,5.866,148.393
C00614=1223.674,162.861,-53.101,-177.826,5.865,148.394
C00615=1223.679,162.612,-53.079,-177.830,5.864,148.394
C00616=1223.684,162.363,-53.057,-177.832,5.863,148.395
C00617=1223.689,162.113,-53.036,-177.834,5.861,148.395
C00618=1223.694,161.865,-53.014,-177.837,5.860,148.396
C00619=1223.699,161.615,-52.992,-177.840,5.859,148.396
C00620=1223.703,161.367,-52.970,-177.842,5.857,148.396
C00621=1223.708,161.118,-52.948,-177.845,5.856,148.397
C00622=1223.713,160.869,-52.927,-177.847,5.854,148.397
C00623=1223.717,160.620,-52.905,-177.850,5.853,148.398
C00624=1223.722,160.370,-52.884,-177.853,5.852,148.398
C00625=1223.727,160.122,-52.862,-177.855,5.851,148.399
C00626=1223.731,159.853,-52.839,-177.857,5.849,148.399
C00627=1223.737,159.584,-52.815,-177.861,5.848,148.400
C00628=1223.741,159.315,-52.792,-177.863,5.846,148.400
C00629=1223.747,159.046,-52.768,-177.866,5.845,148.401
C00630=1223.751,158.796,-52.747,-177.868,5.843,148.401
C00631=1223.756,158.547,-52.725,-177.871,5.843,148.402
C00632=1223.761,158.299,-52.704,-177.874,5.841,148.402
C00633=1223.765,158.049,-52.682,-177.876,5.840,148.402
C00634=1223.770,157.800,-52.661,-177.879,5.838,148.403
C00635=1223.775,157.552,-52.639,-177.881,5.837,148.403
C00636=1223.780,157.302,-52.617,-177.884,5.835,148.404
C00637=1223.784,157.053,-52.597,-177.887,5.834,148.404
C00638=1223.789,156.805,-52.575,-177.889,5.833,148.405
C00639=1223.793,156.555,-52.553,-177.892,5.831,148.405
C00640=1223.798,156.306,-52.532,-177.894,5.831,148.406
C00641=1223.803,156.057,-52.510,-177.897,5.829,148.406
C00642=1223.807,155.808,-52.488,-177.899,5.828,148.406
C00643=1223.813,155.559,-52.467,-177.902,5.826,148.407
C00644=1223.817,155.310,-52.445,-177.904,5.825,148.407
C00645=1223.821,155.061,-52.424,-177.907,5.824,148.408
C00646=1223.826,154.812,-52.403,-177.910,5.823,148.408
C00647=1223.831,154.563,-52.381,-177.912,5.821,148.409
C00648=1223.836,154.314,-52.360,-177.915,5.820,148.409
C00649=1223.841,154.065,-52.338,-177.917,5.818,148.410
C00650=1223.845,153.816,-52.317,-177.920,5.818,148.410
C00651=1223.850,153.567,-52.296,-177.923,5.816,148.411
C00652=1223.855,153.318,-52.275,-177.925,5.815,148.411
C00653=1223.859,153.068,-52.253,-177.927,5.813,148.412
C00654=1223.864,152.820,-52.232,-177.930,5.813,148.412
C00655=1223.869,152.571,-52.211,-177.933,5.811,148.413
C00656=1223.873,152.322,-52.190,-177.935,5.810,148.413
C00657=1223.878,152.072,-52.168,-177.938,5.808,148.414
C00658=1223.883,151.824,-52.147,-177.940,5.807,148.414
C00659=1223.888,151.574,-52.126,-177.943,5.806,148.415
C00660=1223.892,151.326,-52.104,-177.945,5.805,148.415
C00661=1223.897,151.076,-52.083,-177.948,5.803,148.415
C00662=1223.902,150.827,-52.061,-177.951,5.802,148.416
C00663=1223.907,150.578,-52.040,-177.953,5.801,148.416
C00664=1223.911,150.329,-52.020,-177.956,5.800,148.417
C00665=1223.916,150.080,-51.998,-177.959,5.798,148.417
C00666=1223.921,149.831,-51.977,-177.961,5.797,148.418
C00667=1223.925,149.582,-51.956,-177.964,5.796,148.418
C00668=1223.930,149.333,-51.935,-177.966,5.795,148.419
C00669=1223.935,149.084,-51.914,-177.969,5.793,148.419
C00670=1223.939,148.835,-51.893,-177.971,5.792,148.420
C00671=1223.944,148.585,-51.872,-177.974,5.790,148.420
C00672=1223.949,148.337,-51.850,-177.976,5.790,148.421
C00673=1223.953,148.088,-51.830,-177.979,5.789,148.421
C00674=1223.958,147.839,-51.809,-177.982,5.787,148.422
C00675=1223.963,147.590,-51.787,-177.984,5.786,148.422
C00676=1223.967,147.340,-51.766,-177.986,5.784,148.422
C00677=1223.972,147.091,-51.745,-177.989,5.784,148.423
C00678=1223.977,146.842,-51.724,-177.992,5.782,148.423
C00679=1223.982,146.593,-51.703,-177.994,5.781,148.424
C00680=1223.987,146.344,-51.682,-177.997,5.780,148.424
C00681=1223.991,146.095,-51.662,-177.999,5.779,148.425
C00682=1223.996,145.847,-51.640,-178.002,5.777,148.425
C00683=1224.001,145.597,-51.619,-178.004,5.776,148.426
C00684=1224.005,145.348,-51.598,-178.008,5.775,148.426
C00685=1224.010,145.098,-51.577,-178.010,5.774,148.427
C00686=1224.015,144.850,-51.557,-178.012,5.773,148.428
C00687=1224.020,144.601,-51.535,-178.015,5.771,148.428
C00688=1224.024,144.352,-51.515,-178.017,5.770,148.428
C00689=1224.029,144.103,-51.494,-178.020,5.769,148.429
C00690=1224.034,143.853,-51.473,-178.022,5.768,148.429
C00691=1224.038,143.604,-51.452,-178.025,5.766,148.430
C00692=1224.043,143.355,-51.431,-178.028,5.765,148.430
C00693=1224.047,143.106,-51.410,-178.031,5.764,148.431
C00694=1224.053,142.857,-51.389,-178.033,5.763,148.431
C00695=1224.057,142.608,-51.369,-178.035,5.762,148.432
C00696=1224.062,142.359,-51.348,-178.038,5.760,148.432
C00697=1224.067,142.110,-51.328,-178.040,5.759,148.433
C00698=1224.072,141.860,-51.307,-178.043,5.758,148.433
C00699=1224.076,141.612,-51.286,-178.045,5.757,148.434
C00700=1224.081,141.362,-51.265,-178.049,5.756,148.434
C00701=1224.086,141.114,-51.244,-178.051,5.755,148.435
C00702=1224.091,140.865,-51.223,-178.054,5.753,148.435
C00703=1224.095,140.616,-51.203,-178.056,5.752,148.436
C00704=1224.100,140.366,-51.182,-178.058,5.751,148.436
C00705=1224.104,140.117,-51.161,-178.061,5.750,148.437
C00706=1224.109,139.868,-51.141,-178.063,5.749,148.437
C00707=1224.114,139.619,-51.120,-178.067,5.747,148.438
C00708=1224.118,139.370,-51.100,-178.069,5.746,148.438
C00709=1224.123,139.120,-51.079,-178.071,5.746,148.439
C00710=1224.128,138.871,-51.058,-178.074,5.744,148.439
C00711=1224.133,138.622,-51.037,-178.077,5.743,148.440
C00712=1224.137,138.373,-51.017,-178.079,5.741,148.440
C00713=1224.142,138.124,-50.996,-178.081,5.740,148.441
C00714=1224.147,137.875,-50.975,-178.084,5.739,148.441
C00715=1224.152,137.626,-50.955,-178.087,5.738,148.442
C00716=1224.156,137.377,-50.935,-178.089,5.737,148.442
C00717=1224.161,137.127,-50.914,-178.092,5.736,148.443
C00718=1224.166,136.878,-50.894,-178.094,5.735,148.443
C00719=1224.171,136.629,-50.873,-178.097,5.733,148.444
C00720=1224.175,136.380,-50.853,-178.100,5.732,148.444
C00721=1224.180,136.131,-50.832,-178.102,5.731,148.445
C00722=1224.185,135.882,-50.811,-178.105,5.730,148.445
C00723=1224.190,135.633,-50.791,-178.107,5.729,148.446
C00724=1224.194,135.384,-50.771,-178.110,5.728,148.446
C00725=1224.199,135.134,-50.750,-178.112,5.727,148.447
C00726=1224.204,134.885,-50.730,-178.115,5.726,148.447
C00727=1224.209,134.637,-50.710,-178.118,5.724,148.448
C00728=1224.213,134.388,-50.690,-178.120,5.724,148.448
C00729=1224.219,134.139,-50.669,-178.123,5.722,148.449
C00730=1224.223,133.869,-50.647,-178.126,5.721,148.449
C00731=1224.228,133.601,-50.625,-178.128,5.719,148.450
C00732=1224.234,133.332,-50.603,-178.131,5.719,148.450
C00733=1224.238,133.064,-50.581,-178.134,5.717,148.451
C00734=1224.244,132.815,-50.560,-178.136,5.716,148.451
C00735=1224.248,132.565,-50.541,-178.139,5.715,148.452
C00736=1224.253,132.316,-50.520,-178.141,5.714,148.452
C00737=1224.257,132.067,-50.500,-178.144,5.713,148.453
C00738=1224.263,131.817,-50.480,-178.147,5.711,148.453
C00739=1224.267,131.568,-50.459,-178.149,5.711,148.454
C00740=1224.272,131.320,-50.439,-178.151,5.710,148.454
C00741=1224.277,131.071,-50.419,-178.155,5.708,148.455
C00742=1224.282,130.821,-50.399,-178.157,5.707,148.455
C00743=1224.287,130.572,-50.378,-178.160,5.706,148.456
C00744=1224.291,130.324,-50.358,-178.162,5.705,148.456
C00745=1224.296,130.074,-50.338,-178.165,5.704,148.457
C00746=1224.300,129.825,-50.318,-178.167,5.702,148.457
C00747=1224.306,129.575,-50.298,-178.170,5.702,148.458
C00748=1224.310,129.326,-50.277,-178.172,5.701,148.459
C00749=1224.315,129.078,-50.257,-178.175,5.699,148.459
C00750=1224.320,128.828,-50.238,-178.177,5.698,148.460
C00751=1224.324,128.579,-50.217,-178.180,5.698,148.460
C00752=1224.329,128.330,-50.197,-178.183,5.696,148.461
C00753=1224.334,128.081,-50.177,-178.185,5.695,148.461
C00754=1224.339,127.832,-50.156,-178.187,5.694,148.462
C00755=1224.343,127.582,-50.137,-178.190,5.693,148.462
C00756=1224.348,127.334,-50.117,-178.193,5.692,148.463
C00757=1224.353,127.084,-50.097,-178.195,5.691,148.463
C00758=1224.358,126.835,-50.077,-178.198,5.689,148.464
C00759=1224.362,126.586,-50.057,-178.200,5.689,148.464
C00760=1224.367,126.337,-50.037,-178.203,5.687,148.465
C00761=1224.372,126.087,-50.017,-178.206,5.686,148.465
C00762=1224.377,125.839,-49.997,-178.208,5.685,148.466
C00763=1224.381,125.589,-49.977,-178.211,5.684,148.466
C00764=1224.386,125.340,-49.957,-178.214,5.683,148.467
C00765=1224.391,125.091,-49.937,-178.216,5.682,148.467
C00766=1224.396,124.842,-49.916,-178.219,5.681,148.468
C00767=1224.401,124.593,-49.897,-178.221,5.680,148.468
C00768=1224.405,124.344,-49.877,-178.224,5.679,148.469
C00769=1224.410,124.094,-49.857,-178.226,5.678,148.469
C00770=1224.415,123.845,-49.837,-178.229,5.677,148.470
C00771=1224.420,123.596,-49.817,-178.231,5.676,148.470
C00772=1224.425,123.347,-49.798,-178.234,5.675,148.471
C00773=1224.429,123.098,-49.777,-178.236,5.674,148.472
C00774=1224.434,122.848,-49.758,-178.239,5.673,148.472
C00775=1224.439,122.599,-49.738,-178.241,5.672,148.473
C00776=1224.444,122.351,-49.718,-178.244,5.671,148.473
C00777=1224.448,122.101,-49.698,-178.247,5.670,148.474
C00778=1224.453,121.851,-49.679,-178.249,5.669,148.474
C00779=1224.458,121.603,-49.659,-178.252,5.667,148.475
C00780=1224.463,121.354,-49.639,-178.254,5.666,148.475
C00781=1224.468,121.104,-49.619,-178.257,5.666,148.476
C00782=1224.471,120.855,-49.600,-178.259,5.664,148.476
C00783=1224.477,120.606,-49.580,-178.262,5.663,148.477
C00784=1224.482,120.357,-49.561,-178.264,5.662,148.477
C00785=1224.486,120.107,-49.541,-178.267,5.661,148.478
C00786=1224.491,119.858,-49.521,-178.270,5.660,148.479
C00787=1224.496,119.610,-49.501,-178.272,5.659,148.479
C00788=1224.501,119.360,-49.482,-178.275,5.658,148.480
C00789=1224.505,119.111,-49.461,-178.277,5.657,148.480
C00790=1224.511,118.862,-49.442,-178.280,5.656,148.481
C00791=1224.515,118.613,-49.422,-178.282,5.655,148.481
C00792=1224.520,118.363,-49.403,-178.285,5.654,148.482
C00793=1224.525,118.114,-49.384,-178.287,5.653,148.482
C00794=1224.529,117.866,-49.364,-178.290,5.652,148.483
C00795=1224.534,117.616,-49.344,-178.293,5.651,148.483
C00796=1224.539,117.367,-49.325,-178.295,5.650,148.484
C00797=1224.544,117.118,-49.305,-178.298,5.649,148.484
C00798=1224.549,116.868,-49.285,-178.300,5.648,148.485
C00799=1224.554,116.619,-49.266,-178.303,5.647,148.485
C00800=1224.558,116.370,-49.247,-178.306,5.646,148.486
C00801=1224.562,116.121,-49.227,-178.308,5.645,148.487
C00802=1224.568,115.872,-49.207,-178.311,5.644,148.487
C00803=1224.573,115.622,-49.188,-178.313,5.643,148.488
C00804=1224.577,115.373,-49.168,-178.316,5.642,148.488
C00805=1224.583,115.124,-49.149,-178.318,5.641,148.489
C00806=1224.587,114.875,-49.130,-178.321,5.640,148.489
C00807=1224.592,114.626,-49.110,-178.324,5.639,148.490
C00808=1224.597,114.376,-49.091,-178.326,5.638,148.490
C00809=1224.601,114.127,-49.071,-178.329,5.637,148.491
C00810=1224.607,113.878,-49.052,-178.331,5.636,148.491
C00811=1224.611,113.629,-49.033,-178.334,5.635,148.492
C00812=1224.616,113.379,-49.013,-178.336,5.635,148.493
C00813=1224.621,113.130,-48.994,-178.339,5.633,148.493
C00814=1224.626,112.881,-48.974,-178.342,5.632,148.494
C00815=1224.630,112.632,-48.955,-178.344,5.631,148.494
C00816=1224.635,112.382,-48.936,-178.346,5.631,148.495
C00817=1224.640,112.134,-48.916,-178.350,5.629,148.495
C00818=1224.644,111.884,-48.897,-178.352,5.628,148.496
C00819=1224.649,111.635,-48.878,-178.354,5.628,148.496
C00820=1224.654,111.386,-48.858,-178.356,5.627,148.497
C00821=1224.659,111.136,-48.839,-178.360,5.625,148.497
C00822=1224.664,110.888,-48.820,-178.362,5.625,148.498
C00823=1224.669,110.638,-48.800,-178.364,5.624,148.498
C00824=1224.674,110.389,-48.781,-178.367,5.623,148.499
C00825=1224.678,110.140,-48.762,-178.370,5.621,148.500
C00826=1224.683,109.891,-48.742,-178.372,5.621,148.500
C00827=1224.688,109.642,-48.723,-178.375,5.620,148.501
C00828=1224.692,109.392,-48.704,-178.377,5.619,148.501
C00829=1224.698,109.143,-48.686,-178.380,5.618,148.502
C00830=1224.702,108.893,-48.666,-178.382,5.617,148.502
C00831=1224.707,108.645,-48.647,-178.385,5.616,148.503
C00832=1224.712,108.395,-48.628,-178.388,5.616,148.504
C00833=1224.716,108.147,-48.609,-178.390,5.614,148.504
C00834=1224.722,107.877,-48.588,-178.393,5.613,148.505
C00835=1224.727,107.609,-48.568,-178.395,5.612,148.505
C00836=1224.732,107.341,-48.547,-178.399,5.611,148.506
C00837=1224.738,107.072,-48.527,-178.401,5.610,148.506
C00838=1224.742,106.823,-48.508,-178.403,5.609,148.507
C00839=1224.747,106.574,-48.488,-178.407,5.608,148.508
C00840=1224.752,106.325,-48.469,-178.409,5.607,148.508
C00841=1224.756,106.076,-48.450,-178.411,5.606,148.509
C00842=1224.762,105.826,-48.431,-178.414,5.606,148.509
C00843=1224.766,105.577,-48.412,-178.417,5.604,148.510
C00844=1224.771,105.328,-48.393,-178.419,5.603,148.510
C00845=1224.775,105.079,-48.374,-178.422,5.603,148.511
C00846=1224.781,104.829,-48.355,-178.424,5.602,148.511
C00847=1224.785,104.580,-48.336,-178.427,5.601,148.512
C00848=1224.790,104.331,-48.317,-178.430,5.600,148.513
C00849=1224.795,104.082,-48.299,-178.432,5.599,148.513
C00850=1224.800,103.832,-48.279,-178.434,5.598,148.514
C00851=1224.805,103.583,-48.260,-178.437,5.597,148.514
C00852=1224.810,103.334,-48.242,-178.440,5.596,148.515
C00853=1224.815,103.084,-48.222,-178.442,5.595,148.515
C00854=1224.819,102.836,-48.203,-178.445,5.594,148.516
C00855=1224.824,102.586,-48.184,-178.447,5.594,148.516
C00856=1224.829,102.337,-48.166,-178.450,5.593,148.517
C00857=1224.833,102.087,-48.147,-178.452,5.591,148.517
C00858=1224.838,101.838,-48.128,-178.455,5.591,148.518
C00859=1224.843,101.590,-48.109,-178.458,5.590,148.519
C00860=1224.848,101.340,-48.091,-178.460,5.589,148.519
C00861=1224.853,101.091,-48.072,-178.462,5.589,148.520
C00862=1224.858,100.841,-48.053,-178.466,5.587,148.520
C00863=1224.862,100.592,-48.034,-178.468,5.586,148.521
C00864=1224.868,100.343,-48.016,-178.470,5.586,148.522
C00865=1224.872,100.094,-47.997,-178.473,5.585,148.522
C00866=1224.877,99.845,-47.978,-178.475,5.584,148.523
C00867=1224.882,99.595,-47.959,-178.478,5.583,148.523
C00868=1224.886,99.346,-47.940,-178.481,5.582,148.524
C00869=1224.892,99.097,-47.922,-178.483,5.581,148.524
C00870=1224.896,98.848,-47.903,-178.486,5.580,148.525
C00871=1224.901,98.598,-47.885,-178.488,5.580,148.526
C00872=1224.906,98.349,-47.865,-178.490,5.579,148.526
C00873=1224.910,98.100,-47.847,-178.494,5.577,148.527
C00874=1224.916,97.850,-47.828,-178.496,5.577,148.527
C00875=1224.920,97.601,-47.809,-178.498,5.576,148.528
C00876=1224.925,97.352,-47.791,-178.501,5.575,148.528
C00877=1224.930,97.103,-47.772,-178.504,5.575,148.529
C00878=1224.935,96.853,-47.754,-178.506,5.573,148.529
C00879=1224.939,96.604,-47.735,-178.509,5.572,148.530
C00880=1224.945,96.355,-47.716,-178.511,5.572,148.531
C00881=1224.949,96.105,-47.698,-178.514,5.571,148.531
C00882=1224.954,95.857,-47.679,-178.516,5.570,148.532
C00883=1224.960,95.607,-47.661,-178.519,5.569,148.532
C00884=1224.964,95.358,-47.642,-178.522,5.568,148.533
C00885=1224.968,95.109,-47.624,-178.524,5.567,148.534
C00886=1224.973,94.859,-47.606,-178.527,5.567,148.534
C00887=1224.979,94.611,-47.587,-178.529,5.566,148.535
C00888=1224.983,94.361,-47.568,-178.532,5.565,148.535
C00889=1224.988,94.112,-47.550,-178.534,5.564,148.536
C00890=1224.993,93.863,-47.531,-178.537,5.563,148.537
C00891=1224.998,93.613,-47.513,-178.539,5.562,148.537
C00892=1225.003,93.364,-47.495,-178.542,5.561,148.538
C00893=1225.007,93.114,-47.477,-178.545,5.561,148.538
C00894=1225.012,92.865,-47.457,-178.547,5.560,148.539
C00895=1225.017,92.616,-47.439,-178.549,5.559,148.539
C00896=1225.022,92.366,-47.421,-178.553,5.558,148.540
C00897=1225.027,92.118,-47.402,-178.555,5.557,148.540
C00898=1225.031,91.868,-47.384,-178.557,5.556,148.541
C00899=1225.037,91.619,-47.365,-178.560,5.556,148.542
C00900=1225.041,91.369,-47.347,-178.562,5.555,148.542
C00901=1225.046,91.120,-47.329,-178.565,5.554,148.543
C00902=1225.050,90.871,-47.310,-178.567,5.553,148.543
C00903=1225.055,90.622,-47.292,-178.571,5.552,148.544
C00904=1225.061,90.372,-47.274,-178.573,5.551,148.544
C00905=1225.066,90.123,-47.256,-178.575,5.551,148.545
C00906=1225.070,89.873,-47.237,-178.578,5.550,148.546
C00907=1225.075,89.625,-47.219,-178.580,5.549,148.546
C00908=1225.080,89.376,-47.201,-178.583,5.548,148.547
C00909=1225.085,89.126,-47.183,-178.585,5.548,148.548
C00910=1225.090,88.877,-47.164,-178.588,5.547,148.548
C00911=1225.095,88.627,-47.146,-178.591,5.545,148.549
C00912=1225.099,88.378,-47.128,-178.593,5.545,148.549
C00913=1225.104,88.129,-47.110,-178.596,5.544,148.550
C00914=1225.109,87.879,-47.092,-178.598,5.543,148.550
C00915=1225.114,87.631,-47.073,-178.601,5.543,148.551
C00916=1225.118,87.381,-47.055,-178.603,5.542,148.552
C00917=1225.123,87.132,-47.037,-178.606,5.541,148.552
C00918=1225.129,86.882,-47.018,-178.609,5.540,148.553
C00919=1225.134,86.633,-47.000,-178.611,5.539,148.553
C00920=1225.139,86.384,-46.982,-178.614,5.539,148.554
C00921=1225.143,86.134,-46.964,-178.616,5.538,148.554
C00922=1225.148,85.885,-46.946,-178.619,5.537,148.555
C00923=1225.153,85.636,-46.928,-178.621,5.536,148.556
C00924=1225.158,85.387,-46.910,-178.624,5.536,148.556
C00925=1225.163,85.137,-46.892,-178.626,5.535,148.557
C00926=1225.167,84.888,-46.874,-178.629,5.534,148.557
C00927=1225.172,84.639,-46.856,-178.632,5.533,148.558
C00928=1225.177,84.389,-46.838,-178.634,5.532,148.559
C00929=1225.182,84.140,-46.820,-178.637,5.531,148.559
C00930=1225.187,83.891,-46.802,-178.639,5.531,148.560
C00931=1225.191,83.642,-46.784,-178.642,5.530,148.560
C00932=1225.196,83.393,-46.766,-178.644,5.530,148.561
C00933=1225.201,83.143,-46.748,-178.647,5.529,148.562
C00934=1225.206,82.894,-46.730,-178.649,5.528,148.562
C00935=1225.210,82.644,-46.712,-178.652,5.527,148.563
C00936=1225.216,82.394,-46.694,-178.654,5.526,148.563
C00937=1225.221,82.145,-46.676,-178.657,5.525,148.564
C00938=1225.226,81.877,-46.657,-178.660,5.524,148.565
C00939=1225.231,81.609,-46.638,-178.662,5.524,148.565
C00940=1225.236,81.341,-46.618,-178.665,5.523,148.566
C00941=1225.242,81.071,-46.599,-178.668,5.522,148.567
C00942=1225.246,80.822,-46.581,-178.671,5.521,148.567
C00943=1225.251,80.573,-46.563,-178.673,5.521,148.568
C00944=1225.256,80.324,-46.545,-178.676,5.520,148.568
C00945=1225.261,80.075,-46.527,-178.678,5.519,148.569
C00946=1225.266,79.826,-46.510,-178.681,5.519,148.570
C00947=1225.271,79.576,-46.492,-178.683,5.518,148.570
C00948=1225.276,79.327,-46.474,-178.686,5.517,148.571
C00949=1225.281,79.078,-46.456,-178.688,5.516,148.571
C00950=1225.286,78.828,-46.438,-178.691,5.516,148.572
C00951=1225.291,78.579,-46.420,-178.693,5.515,148.573
C00952=1225.296,78.329,-46.403,-178.696,5.513,148.573
C00953=1225.301,78.080,-46.385,-178.699,5.513,148.574
C00954=1225.305,77.831,-46.368,-178.701,5.512,148.574
C00955=1225.310,77.582,-46.350,-178.704,5.512,148.575
C00956=1225.315,77.332,-46.332,-178.706,5.511,148.575
C00957=1225.320,77.083,-46.314,-178.709,5.510,148.576
C00958=1225.324,76.833,-46.296,-178.711,5.510,148.577
C00959=1225.330,76.584,-46.279,-178.714,5.509,148.577
C00960=1225.334,76.334,-46.261,-178.716,5.508,148.578
C00961=1225.339,76.086,-46.244,-178.719,5.507,148.579
C00962=1225.344,75.836,-46.226,-178.721,5.507,148.579
C00963=1225.349,75.587,-46.208,-178.724,5.506,148.580
C00964=1225.354,75.337,-46.190,-178.727,5.506,148.581
C00965=1225.359,75.088,-46.172,-178.729,5.505,148.581
C00966=1225.363,74.839,-46.156,-178.732,5.503,148.582
C00967=1225.368,74.590,-46.138,-178.735,5.503,148.582
C00968=1225.373,74.340,-46.120,-178.737,5.502,148.583
C00969=1225.378,74.091,-46.102,-178.739,5.501,148.583
C00970=1225.383,73.841,-46.084,-178.742,5.501,148.584
C00971=1225.387,73.592,-46.068,-178.745,5.500,148.585
C00972=1225.393,73.344,-46.050,-178.747,5.499,148.585
C00973=1225.398,73.094,-46.033,-178.750,5.499,148.586
C00974=1225.403,72.845,-46.015,-178.752,5.498,148.586
C00975=1225.407,72.596,-45.998,-178.755,5.497,148.587
C00976=1225.413,72.346,-45.980,-178.757,5.497,148.588
C00977=1225.417,72.097,-45.962,-178.760,5.496,148.588
C00978=1225.423,71.847,-45.945,-178.762,5.495,148.589
C00979=1225.427,71.598,-45.928,-178.765,5.495,148.590
C00980=1225.432,71.348,-45.910,-178.767,5.494,148.590
C00981=1225.437,71.099,-45.892,-178.770,5.494,148.591
C00982=1225.441,70.850,-45.876,-178.773,5.493,148.591
C00983=1225.446,70.600,-45.858,-178.775,5.492,148.592
C00984=1225.452,70.351,-45.840,-178.777,5.491,148.593
C00985=1225.456,70.101,-45.822,-178.780,5.491,148.593
C00986=1225.461,69.852,-45.806,-178.783,5.489,148.594
C00987=1225.466,69.603,-45.788,-178.786,5.489,148.595
C00988=1225.471,69.353,-45.771,-178.788,5.488,148.595
C00989=1225.476,69.105,-45.754,-178.791,5.487,148.596
C00990=1225.481,68.855,-45.736,-178.793,5.487,148.596
C00991=1225.486,68.605,-45.719,-178.796,5.486,148.597
C00992=1225.490,68.356,-45.702,-178.798,5.486,148.598
C00993=1225.496,68.107,-45.684,-178.801,5.485,148.598
C00994=1225.500,67.858,-45.667,-178.803,5.484,148.599
C00995=1225.505,67.608,-45.650,-178.806,5.483,148.599
C00996=1225.510,67.358,-45.632,-178.808,5.483,148.600
C00997=1225.514,67.109,-45.615,-178.811,5.482,148.601
C00998=1225.520,66.860,-45.598,-178.813,5.481,148.601
C00999=1225.525,66.611,-45.580,-178.816,5.481,148.602
C01000=1225.530,66.362,-45.564,-178.819,5.480,148.602
C01001=1225.535,66.112,-45.546,-178.821,5.480,148.603
C01002=1225.539,65.863,-45.529,-178.824,5.479,148.604
C01003=1225.544,65.613,-45.512,-178.826,5.478,148.604
C01004=1225.549,65.364,-45.495,-178.829,5.478,148.605
C01005=1225.554,65.115,-45.477,-178.831,5.477,148.606
C01006=1225.560,64.865,-45.460,-178.834,5.476,148.606
C01007=1225.564,64.616,-45.443,-178.836,5.476,148.607
C01008=1225.569,64.366,-45.426,-178.839,5.475,148.608
C01009=1225.573,64.117,-45.409,-178.841,5.474,148.608
C01010=1225.579,63.867,-45.391,-178.844,5.474,148.609
C01011=1225.584,63.619,-45.375,-178.846,5.473,148.609
C01012=1225.589,63.369,-45.358,-178.849,5.473,148.610
C01013=1225.593,63.120,-45.341,-178.852,5.472,148.611
C01014=1225.598,62.870,-45.323,-178.854,5.471,148.611
C01015=1225.603,62.621,-45.307,-178.857,5.470,148.612
C01016=1225.609,62.372,-45.290,-178.859,5.470,148.612
C01017=1225.613,62.123,-45.272,-178.862,5.469,148.613
C01018=1225.618,61.873,-45.255,-178.864,5.469,148.614
C01019=1225.622,61.623,-45.238,-178.867,5.468,148.614
C01020=1225.628,61.374,-45.221,-178.869,5.467,148.615
C01021=1225.633,61.125,-45.205,-178.872,5.467,148.615
C01022=1225.638,60.876,-45.187,-178.874,5.466,148.616
C01023=1225.642,60.626,-45.170,-178.877,5.466,148.617
C01024=1225.647,60.376,-45.153,-178.880,5.465,148.617
C01025=1225.652,60.127,-45.136,-178.882,5.464,148.618
C01026=1225.658,59.878,-45.119,-178.884,5.463,148.619
C01027=1225.662,59.628,-45.103,-178.887,5.463,148.619
C01028=1225.667,59.379,-45.086,-178.890,5.462,148.620
C01029=1225.672,59.129,-45.069,-178.892,5.462,148.621
C01030=1225.677,58.881,-45.052,-178.895,5.461,148.621
C01031=1225.682,58.631,-45.034,-178.898,5.461,148.622
C01032=1225.686,58.382,-45.018,-178.900,5.460,148.622
C01033=1225.692,58.132,-45.001,-178.902,5.459,148.623
C01034=1225.697,57.883,-44.984,-178.905,5.459,148.624
C01035=1225.701,57.634,-44.968,-178.908,5.458,148.624
C01036=1225.706,57.384,-44.950,-178.910,5.457,148.625
C01037=1225.711,57.135,-44.934,-178.913,5.457,148.626
C01038=1225.717,56.885,-44.917,-178.915,5.456,148.626
C01039=1225.721,56.636,-44.900,-178.918,5.455,148.627
C01040=1225.726,56.386,-44.883,-178.920,5.455,148.627
C01041=1225.731,56.137,-44.866,-178.923,5.454,148.628
C01042=1225.736,55.869,-44.848,-178.926,5.454,148.629
C01043=1225.741,55.601,-44.831,-178.928,5.453,148.629
C01044=1225.747,55.331,-44.813,-178.931,5.452,148.630
C01045=1225.752,55.063,-44.795,-178.934,5.452,148.631
C01046=1225.757,54.814,-44.778,-178.936,5.451,148.631
C01047=1225.762,54.564,-44.761,-178.939,5.451,148.632
C01048=1225.767,54.315,-44.745,-178.941,5.450,148.633
C01049=1225.772,54.065,-44.727,-178.944,5.450,148.633
C01050=1225.777,53.816,-44.711,-178.947,5.449,148.634
C01051=1225.782,53.567,-44.694,-178.949,5.448,148.635
C01052=1225.786,53.318,-44.678,-178.952,5.448,148.635
C01053=1225.791,53.068,-44.661,-178.954,5.447,148.636
C01054=1225.797,52.819,-44.644,-178.957,5.446,148.637
C01055=1225.801,52.569,-44.628,-178.959,5.446,148.637
C01056=1225.807,52.319,-44.611,-178.962,5.445,148.638
C01057=1225.812,52.070,-44.595,-178.965,5.445,148.639
C01058=1225.816,51.821,-44.578,-178.967,5.444,148.639
C01059=1225.821,51.571,-44.561,-178.969,5.443,148.640
C01060=1225.826,51.323,-44.545,-178.972,5.443,148.640
C01061=1225.831,51.073,-44.528,-178.974,5.443,148.641
C01062=1225.836,50.823,-44.512,-178.977,5.442,148.642
C01063=1225.841,50.574,-44.496,-178.979,5.442,148.642
C01064=1225.845,50.325,-44.479,-178.982,5.441,148.643
C01065=1225.851,50.075,-44.462,-178.984,5.440,148.643
C01066=1225.856,49.826,-44.445,-178.987,5.440,148.644
C01067=1225.860,49.576,-44.429,-178.989,5.439,148.645
C01068=1225.865,49.327,-44.413,-178.992,5.439,148.645
C01069=1225.870,49.078,-44.396,-178.995,5.438,148.646
C01070=1225.876,48.828,-44.379,-178.997,5.437,148.647
C01071=1225.880,48.579,-44.363,-179.000,5.437,148.648
C01072=1225.885,48.329,-44.347,-179.003,5.436,148.648
C01073=1225.890,48.080,-44.331,-179.005,5.435,148.649
C01074=1225.895,47.831,-44.314,-179.007,5.435,148.649
C01075=1225.900,47.581,-44.298,-179.010,5.434,148.650
C01076=1225.905,47.331,-44.281,-179.012,5.435,148.651
C01077=1225.910,47.083,-44.265,-179.015,5.434,148.651
C01078=1225.915,46.833,-44.248,-179.017,5.433,148.652
C01079=1225.920,46.583,-44.232,-179.020,5.433,148.653
C01080=1225.925,46.334,-44.216,-179.023,5.432,148.653
C01081=1225.929,46.085,-44.199,-179.025,5.431,148.654
C01082=1225.934,45.835,-44.184,-179.027,5.431,148.654
C01083=1225.939,45.586,-44.167,-179.030,5.430,148.655
C01084=1225.945,45.336,-44.151,-179.033,5.430,148.656
C01085=1225.950,45.087,-44.134,-179.035,5.429,148.656
C01086=1225.955,44.838,-44.118,-179.038,5.429,148.657
C01087=1225.959,44.588,-44.102,-179.041,5.428,148.658
C01088=1225.964,44.339,-44.085,-179.043,5.427,148.658
C01089=1225.969,44.090,-44.069,-179.045,5.428,148.659
C01090=1225.974,43.840,-44.053,-179.048,5.427,148.660
C01091=1225.979,43.591,-44.037,-179.050,5.426,148.660
C01092=1225.984,43.341,-44.021,-179.053,5.426,148.661
C01093=1225.989,43.092,-44.004,-179.055,5.425,148.662
C01094=1225.993,42.842,-43.988,-179.058,5.425,148.662
C01095=1225.999,42.593,-43.972,-179.061,5.424,148.663
C01096=1226.003,42.343,-43.955,-179.063,5.423,148.664
C01097=1226.008,42.094,-43.940,-179.066,5.423,148.664
C01098=1226.013,41.845,-43.923,-179.069,5.422,148.665
C01099=1226.018,41.595,-43.908,-179.071,5.421,148.665
C01100=1226.023,41.346,-43.891,-179.073,5.422,148.666
C01101=1226.028,41.096,-43.875,-179.076,5.421,148.667
C01102=1226.033,40.847,-43.859,-179.078,5.421,148.667
C01103=1226.038,40.597,-43.843,-179.081,5.420,148.668
C01104=1226.043,40.349,-43.827,-179.083,5.419,148.669
C01105=1226.048,40.098,-43.811,-179.086,5.419,148.669
C01106=1226.053,39.850,-43.794,-179.089,5.418,148.670
C01107=1226.058,39.600,-43.778,-179.091,5.418,148.671
C01108=1226.063,39.350,-43.763,-179.094,5.417,148.671
C01109=1226.068,39.101,-43.746,-179.096,5.416,148.672
C01110=1226.073,38.851,-43.731,-179.098,5.417,148.673
C01111=1226.078,38.602,-43.714,-179.101,5.416,148.673
C01112=1226.083,38.352,-43.698,-179.103,5.415,148.674
C01113=1226.088,38.103,-43.683,-179.106,5.415,148.675
C01114=1226.093,37.854,-43.666,-179.109,5.414,148.675
C01115=1226.098,37.604,-43.651,-179.111,5.414,148.676
C01116=1226.103,37.355,-43.634,-179.114,5.413,148.677
C01117=1226.108,37.105,-43.618,-179.117,5.413,148.677
C01118=1226.113,36.856,-43.603,-179.119,5.412,148.678
C01119=1226.118,36.606,-43.586,-179.121,5.412,148.678
C01120=1226.123,36.357,-43.570,-179.124,5.411,148.679
C01121=1226.127,36.107,-43.555,-179.126,5.411,148.680
C01122=1226.132,35.858,-43.539,-179.129,5.410,148.680
C01123=1226.138,35.609,-43.523,-179.131,5.410,148.681
C01124=1226.143,35.359,-43.507,-179.134,5.409,148.682
C01125=1226.148,35.110,-43.491,-179.137,5.409,148.683
C01126=1226.152,34.860,-43.475,-179.139,5.408,148.683
C01127=1226.158,34.611,-43.459,-179.141,5.408,148.684
C01128=1226.163,34.362,-43.443,-179.144,5.408,148.685
C01129=1226.167,34.112,-43.428,-179.147,5.407,148.685
C01130=1226.172,33.863,-43.412,-179.149,5.407,148.686
C01131=1226.177,33.612,-43.396,-179.152,5.406,148.686
C01132=1226.182,33.364,-43.380,-179.154,5.405,148.687
C01133=1226.188,33.114,-43.364,-179.157,5.405,148.688
C01134=1226.192,32.864,-43.348,-179.159,5.405,148.688
C01135=1226.197,32.615,-43.333,-179.162,5.404,148.689
C01136=1226.202,32.366,-43.318,-179.164,5.404,148.690
C01137=1226.207,32.116,-43.301,-179.167,5.403,148.690
C01138=1226.212,31.867,-43.285,-179.169,5.403,148.691
C01139=1226.218,31.617,-43.270,-179.172,5.402,148.692
C01140=1226.222,31.368,-43.255,-179.175,5.402,148.692
C01141=1226.227,31.118,-43.239,-179.177,5.401,148.693
C01142=1226.232,30.869,-43.223,-179.179,5.401,148.694
C01143=1226.237,30.619,-43.207,-179.182,5.401,148.694
C01144=1226.242,30.370,-43.192,-179.184,5.400,148.695
C01145=1226.247,30.121,-43.176,-179.187,5.399,148.696
C01146=1226.253,29.852,-43.159,-179.190,5.399,148.697
C01147=1226.258,29.583,-43.142,-179.193,5.399,148.697
C01148=1226.263,29.315,-43.125,-179.195,5.398,148.698
C01149=1226.268,29.046,-43.109,-179.198,5.398,148.699
C01150=1226.273,28.797,-43.093,-179.201,5.397,148.699
C01151=1226.278,28.547,-43.077,-179.203,5.396,148.700
C01152=1226.283,28.298,-43.062,-179.205,5.397,148.701
C01153=1226.288,28.049,-43.046,-179.208,5.396,148.701
C01154=1226.293,27.799,-43.031,-179.211,5.396,148.702
C01155=1226.298,27.549,-43.015,-179.213,5.395,148.703
C01156=1226.303,27.300,-43.000,-179.216,5.395,148.703
C01157=1226.308,27.051,-42.984,-179.218,5.394,148.704
C01158=1226.314,26.801,-42.968,-179.221,5.393,148.704
C01159=1226.318,26.551,-42.953,-179.223,5.393,148.705
C01160=1226.323,26.302,-42.938,-179.225,5.393,148.706
C01161=1226.329,26.053,-42.922,-179.228,5.392,148.706
C01162=1226.333,25.803,-42.907,-179.231,5.392,148.707
C01163=1226.338,25.553,-42.891,-179.233,5.391,148.708
C01164=1226.343,25.304,-42.875,-179.236,5.391,148.708
C01165=1226.348,25.055,-42.860,-179.238,5.391,148.709
C01166=1226.353,24.805,-42.845,-179.241,5.390,148.710
C01167=1226.357,24.556,-42.829,-179.243,5.390,148.711
C01168=1226.363,24.306,-42.814,-179.246,5.389,148.711
C01169=1226.368,24.057,-42.798,-179.249,5.389,148.712
C01170=1226.373,23.808,-42.783,-179.251,5.388,148.713
C01171=1226.378,23.558,-42.767,-179.253,5.388,148.713
C01172=1226.383,23.308,-42.752,-179.256,5.388,148.714
C01173=1226.388,23.059,-42.737,-179.259,5.387,148.715
C01174=1226.393,22.809,-42.722,-179.261,5.386,148.715
C01175=1226.398,22.560,-42.707,-179.263,5.386,148.716
C01176=1226.403,22.310,-42.691,-179.266,5.386,148.716
C01177=1226.407,22.061,-42.676,-179.268,5.386,148.717
C01178=1226.413,21.811,-42.660,-179.271,5.385,148.718
C01179=1226.418,21.562,-42.645,-179.273,5.385,148.718
C01180=1226.423,21.313,-42.630,-179.276,5.384,148.719
C01181=1226.428,21.063,-42.614,-179.279,5.383,148.720
C01182=1226.433,20.813,-42.600,-179.281,5.384,148.721
C01183=1226.438,20.564,-42.584,-179.284,5.383,148.721
C01184=1226.443,20.315,-42.569,-179.286,5.383,148.722
C01185=1226.448,20.065,-42.553,-179.289,5.382,148.723
C01186=1226.453,19.816,-42.538,-179.291,5.382,148.723
C01187=1226.457,19.566,-42.522,-179.294,5.382,148.724
C01188=1226.462,19.316,-42.508,-179.296,5.381,148.725
C01189=1226.468,19.067,-42.493,-179.299,5.381,148.725
C01190=1226.472,18.818,-42.478,-179.301,5.380,148.726
C01191=1226.478,18.568,-42.462,-179.304,5.380,148.727
C01192=1226.483,18.319,-42.448,-179.306,5.380,148.727
C01193=1226.488,18.069,-42.432,-179.309,5.379,148.728
C01194=1226.492,17.820,-42.417,-179.311,5.379,148.729
C01195=1226.498,17.570,-42.401,-179.314,5.378,148.729
C01196=1226.503,17.320,-42.387,-179.316,5.377,148.730
C01197=1226.508,17.071,-42.371,-179.319,5.377,148.731
C01198=1226.513,16.822,-42.356,-179.321,5.377,148.731
C01199=1226.518,16.573,-42.341,-179.324,5.377,148.732
C01200=1226.523,16.323,-42.326,-179.326,5.376,148.733
C01201=1226.528,16.074,-42.311,-179.329,5.376,148.733
C01202=1226.532,15.824,-42.295,-179.331,5.376,148.734
C01203=1226.537,15.574,-42.281,-179.334,5.375,148.735
C01204=1226.543,15.324,-42.266,-179.336,5.375,148.735
C01205=1226.547,15.075,-42.251,-179.339,5.374,148.736
C01206=1226.553,14.825,-42.236,-179.342,5.374,148.737
C01207=1226.558,14.576,-42.221,-179.344,5.374,148.737
C01208=1226.562,14.327,-42.206,-179.346,5.373,148.738
C01209=1226.568,14.077,-42.191,-179.349,5.373,148.739
C01210=1226.573,13.828,-42.176,-179.352,5.372,148.739
C01211=1226.578,13.578,-42.161,-179.354,5.372,148.740
C01212=1226.583,13.329,-42.146,-179.356,5.372,148.741
C01213=1226.587,13.079,-42.131,-179.359,5.372,148.741
C01214=1226.593,12.829,-42.116,-179.362,5.371,148.742
C01215=1226.597,12.580,-42.101,-179.364,5.371,148.743
C01216=1226.602,12.330,-42.087,-179.367,5.370,148.744
C01217=1226.608,12.081,-42.071,-179.369,5.370,148.744
C01218=1226.613,11.831,-42.057,-179.372,5.370,148.745
C01219=1226.617,11.582,-42.042,-179.374,5.369,148.746
C01220=1226.623,11.333,-42.026,-179.377,5.369,148.746
C01221=1226.628,11.083,-42.012,-179.379,5.369,148.747
C01222=1226.632,10.834,-41.997,-179.382,5.368,148.748
C01223=1226.638,10.584,-41.982,-179.384,5.368,148.748
C01224=1226.643,10.335,-41.967,-179.387,5.367,148.749
C01225=1226.648,10.085,-41.953,-179.390,5.367,148.750
C01226=1226.653,9.836,-41.937,-179.391,5.367,148.750
C01227=1226.658,9.586,-41.923,-179.394,5.366,148.751
C01228=1226.663,9.337,-41.908,-179.397,5.366,148.752
C01229=1226.668,9.087,-41.894,-179.399,5.365,148.752
C01230=1226.673,8.838,-41.878,-179.401,5.365,148.753
C01231=1226.678,8.588,-41.864,-179.404,5.365,148.754
C01232=1226.683,8.338,-41.849,-179.407,5.364,148.754
C01233=1226.688,8.089,-41.834,-179.409,5.364,148.755
C01234=1226.693,7.839,-41.820,-179.411,5.364,148.756
C01235=1226.698,7.590,-41.805,-179.414,5.364,148.756
C01236=1226.703,7.340,-41.790,-179.417,5.363,148.757
C01237=1226.708,7.091,-41.775,-179.419,5.363,148.758
C01238=1226.713,6.841,-41.760,-179.422,5.362,148.758
C01239=1226.718,6.592,-41.746,-179.424,5.362,148.759
C01240=1226.723,6.343,-41.731,-179.427,5.362,148.760
C01241=1226.728,6.093,-41.717,-179.429,5.361,148.760
C01242=1226.733,5.843,-41.702,-179.432,5.361,148.761
C01243=1226.738,5.594,-41.687,-179.434,5.361,148.762
C01244=1226.743,5.344,-41.673,-179.437,5.360,148.763
C01245=1226.748,5.095,-41.658,-179.439,5.360,148.763
C01246=1226.753,4.845,-41.643,-179.442,5.359,148.764
C01247=1226.758,4.595,-41.629,-179.444,5.360,148.765
C01248=1226.763,4.346,-41.614,-179.447,5.359,148.765
C01249=1226.769,4.097,-41.600,-179.449,5.359,148.766
C01250=1226.774,3.828,-41.584,-179.452,5.358,148.767
C01251=1226.779,3.559,-41.569,-179.455,5.358,148.767
C01252=1226.785,3.290,-41.553,-179.457,5.358,148.768
C01253=1226.790,3.021,-41.537,-179.460,5.358,148.769
C01254=1226.795,2.771,-41.523,-179.463,5.357,148.770
C01255=1226.800,2.522,-41.508,-179.465,5.357,148.770
C01256=1226.805,2.272,-41.493,-179.468,5.356,148.771
C01257=1226.810,2.023,-41.479,-179.470,5.356,148.772
C01258=1226.815,1.773,-41.464,-179.473,5.356,148.772
C01259=1226.820,1.524,-41.449,-179.475,5.355,148.773
C01260=1226.826,1.275,-41.435,-179.478,5.355,148.774
C01261=1226.830,1.025,-41.421,-179.480,5.355,148.774
C01262=1226.835,0.775,-41.407,-179.483,5.355,148.775
C01263=1226.840,0.526,-41.393,-179.485,5.354,148.776
C01264=1226.845,0.276,-41.378,-179.488,5.354,148.777
C01265=1226.850,0.027,-41.363,-179.490,5.354,148.777
C01266=1226.855,-0.223,-41.349,-179.493,5.353,148.778
C01267=1226.860,-0.473,-41.335,-179.495,5.353,148.779
C01268=1226.865,-0.722,-41.321,-179.497,5.353,148.779
C01269=1226.870,-0.971,-41.307,-179.500,5.353,148.780
C01270=1226.876,-1.221,-41.291,-179.503,5.352,148.781
C01271=1226.881,-1.471,-41.277,-179.505,5.352,148.781
C01272=1226.886,-1.720,-41.262,-179.507,5.352,148.782
C01273=1226.891,-1.970,-41.248,-179.510,5.351,148.783
C01274=1226.896,-2.220,-41.234,-179.513,5.351,148.783
C01275=1226.901,-2.469,-41.220,-179.515,5.350,148.784
C01276=1226.906,-2.718,-41.206,-179.517,5.351,148.785
C01277=1226.911,-2.968,-41.191,-179.520,5.350,148.785
C01278=1226.916,-3.217,-41.176,-179.523,5.350,148.786
C01279=1226.921,-3.467,-41.162,-179.525,5.350,148.787
C01280=1226.926,-3.717,-41.148,-179.527,5.349,148.788
C01281=1226.931,-3.966,-41.134,-179.530,5.349,148.788
C01282=1226.936,-4.215,-41.120,-179.533,5.348,148.789
C01283=1226.941,-4.465,-41.105,-179.535,5.349,148.790
C01284=1226.946,-4.715,-41.091,-179.538,5.348,148.790
C01285=1226.951,-4.964,-41.077,-179.540,5.348,148.791
C01286=1226.957,-5.213,-41.063,-179.543,5.347,148.792
C01287=1226.962,-5.463,-41.049,-179.545,5.347,148.792
C01288=1226.966,-5.713,-41.034,-179.548,5.347,148.793
C01289=1226.971,-5.963,-41.020,-179.550,5.346,148.794
C01290=1226.976,-6.212,-41.006,-179.552,5.347,148.794
C01291=1226.981,-6.461,-40.992,-179.555,5.346,148.795
C01292=1226.986,-6.711,-40.978,-179.558,5.346,148.796
C01293=1226.991,-6.960,-40.964,-179.560,5.345,148.797
C01294=1226.996,-7.210,-40.950,-179.562,5.345,148.797
C01295=1227.002,-7.459,-40.936,-179.565,5.345,148.798
C01296=1227.007,-7.709,-40.921,-179.568,5.344,148.799
C01297=1227.012,-7.959,-40.907,-179.570,5.345,148.799
C01298=1227.016,-8.208,-40.893,-179.572,5.344,148.800
C01299=1227.021,-8.458,-40.879,-179.575,5.344,148.801
C01300=1227.027,-8.707,-40.865,-179.577,5.344,148.801
C01301=1227.032,-8.957,-40.852,-179.580,5.343,148.802
C01302=1227.036,-9.207,-40.837,-179.582,5.343,148.803
C01303=1227.041,-9.456,-40.823,-179.585,5.342,148.803
C01304=1227.047,-9.705,-40.809,-179.587,5.343,148.804
C01305=1227.052,-9.955,-40.795,-179.590,5.342,148.805
C01306=1227.057,-10.205,-40.781,-179.592,5.342,148.806
C01307=1227.062,-10.454,-40.767,-179.595,5.342,148.806
C01308=1227.067,-10.703,-40.753,-179.597,5.341,148.807
C01309=1227.072,-10.954,-40.740,-179.600,5.341,148.808
C01310=1227.077,-11.203,-40.725,-179.602,5.341,148.808
C01311=1227.082,-11.452,-40.711,-179.605,5.341,148.809
C01312=1227.087,-11.702,-40.697,-179.607,5.340,148.810
C01313=1227.092,-11.952,-40.683,-179.610,5.340,148.810
C01314=1227.097,-12.200,-40.669,-179.612,5.340,148.811
C01315=1227.102,-12.451,-40.656,-179.615,5.339,148.812
C01316=1227.107,-12.700,-40.642,-179.617,5.339,148.812
C01317=1227.112,-12.950,-40.627,-179.619,5.339,148.813
C01318=1227.118,-13.199,-40.613,-179.622,5.339,148.814
C01319=1227.122,-13.449,-40.600,-179.625,5.338,148.815
C01320=1227.127,-13.699,-40.586,-179.627,5.338,148.815
C01321=1227.133,-13.948,-40.572,-179.629,5.338,148.816
C01322=1227.138,-14.198,-40.558,-179.632,5.337,148.817
C01323=1227.143,-14.447,-40.544,-179.634,5.338,148.817
C01324=1227.148,-14.697,-40.531,-179.637,5.337,148.818
C01325=1227.153,-14.946,-40.517,-179.639,5.337,148.819
C01326=1227.158,-15.196,-40.503,-179.642,5.336,148.819
C01327=1227.164,-15.446,-40.489,-179.644,5.336,148.820
C01328=1227.168,-15.695,-40.476,-179.647,5.336,148.821
C01329=1227.173,-15.945,-40.461,-179.650,5.335,148.821
C01330=1227.178,-16.194,-40.448,-179.652,5.336,148.822
C01331=1227.183,-16.444,-40.435,-179.654,5.335,148.823
C01332=1227.189,-16.693,-40.421,-179.657,5.335,148.824
C01333=1227.193,-16.943,-40.406,-179.659,5.335,148.824
C01334=1227.199,-17.193,-40.393,-179.662,5.335,148.825
C01335=1227.204,-17.442,-40.379,-179.664,5.334,148.826
C01336=1227.209,-17.691,-40.365,-179.666,5.334,148.826
C01337=1227.214,-17.942,-40.352,-179.669,5.334,148.827
C01338=1227.219,-18.190,-40.338,-179.672,5.333,148.828
C01339=1227.224,-18.441,-40.325,-179.674,5.334,148.828
C01340=1227.229,-18.690,-40.311,-179.676,5.333,148.829
C01341=1227.234,-18.939,-40.297,-179.679,5.333,148.830
C01342=1227.239,-19.189,-40.284,-179.681,5.333,148.830
C01343=1227.244,-19.438,-40.270,-179.684,5.332,148.831
C01344=1227.249,-19.688,-40.257,-179.687,5.332,148.832
C01345=1227.255,-19.937,-40.243,-179.689,5.332,148.833
C01346=1227.259,-20.187,-40.229,-179.691,5.332,148.833
C01347=1227.264,-20.437,-40.216,-179.694,5.331,148.834
C01348=1227.270,-20.686,-40.202,-179.696,5.331,148.835
C01349=1227.275,-20.937,-40.188,-179.699,5.331,148.835
C01350=1227.280,-21.185,-40.175,-179.701,5.330,148.836
C01351=1227.285,-21.436,-40.161,-179.703,5.331,148.837
C01352=1227.290,-21.684,-40.148,-179.706,5.330,148.837
C01353=1227.295,-21.935,-40.134,-179.709,5.330,148.838
C01354=1227.300,-22.204,-40.119,-179.711,5.330,148.839
C01355=1227.306,-22.473,-40.105,-179.714,5.330,148.840
C01356=1227.311,-22.742,-40.090,-179.717,5.329,148.840
C01357=1227.317,-23.012,-40.076,-179.719,5.329,148.841
C01358=1227.322,-23.262,-40.062,-179.721,5.329,148.842
C01359=1227.327,-23.511,-40.049,-179.724,5.329,148.843
C01360=1227.332,-23.761,-40.035,-179.727,5.328,148.843
C01361=1227.337,-24.010,-40.022,-179.729,5.329,148.844
C01362=1227.342,-24.260,-40.008,-179.731,5.328,148.845
C01363=1227.347,-24.509,-39.995,-179.734,5.328,148.845
C01364=1227.352,-24.759,-39.981,-179.736,5.328,148.846
C01365=1227.358,-25.008,-39.968,-179.739,5.327,148.847
C01366=1227.362,-25.258,-39.955,-179.741,5.327,148.847
C01367=1227.368,-25.507,-39.941,-179.744,5.327,148.848
C01368=1227.373,-25.757,-39.928,-179.746,5.327,148.849
C01369=1227.378,-26.006,-39.914,-179.749,5.326,148.850
C01370=1227.383,-26.256,-39.901,-179.751,5.327,148.850
C01371=1227.388,-26.506,-39.888,-179.754,5.326,148.851
C01372=1227.393,-26.755,-39.874,-179.757,5.326,148.852
C01373=1227.399,-27.005,-39.861,-179.759,5.326,148.853
C01374=1227.403,-27.255,-39.848,-179.762,5.326,148.853
C01375=1227.409,-27.504,-39.834,-179.764,5.325,148.854
C01376=1227.413,-27.754,-39.821,-179.766,5.325,148.855
C01377=1227.419,-28.004,-39.808,-179.769,5.325,148.855
C01378=1227.423,-28.253,-39.794,-179.771,5.325,148.856
C01379=1227.428,-28.502,-39.782,-179.774,5.325,148.857
C01380=1227.434,-28.753,-39.768,-179.776,5.324,148.857
C01381=1227.438,-29.001,-39.755,-179.778,5.325,148.858
C01382=1227.444,-29.252,-39.741,-179.781,5.324,148.859
C01383=1227.449,-29.501,-39.729,-179.784,5.324,148.860
C01384=1227.454,-29.751,-39.715,-179.786,5.324,148.860
C01385=1227.459,-30.000,-39.702,-179.788,5.323,148.861
C01386=1227.465,-30.250,-39.689,-179.791,5.323,148.862
C01387=1227.469,-30.500,-39.676,-179.793,5.323,148.862
C01388=1227.474,-30.748,-39.662,-179.796,5.323,148.863
C01389=1227.479,-30.999,-39.649,-179.798,5.323,148.864
C01390=1227.484,-31.248,-39.636,-179.801,5.323,148.864
C01391=1227.490,-31.498,-39.623,-179.803,5.322,148.865
C01392=1227.495,-31.747,-39.609,-179.805,5.322,148.866
C01393=1227.500,-31.996,-39.597,-179.808,5.322,148.866
C01394=1227.505,-32.247,-39.583,-179.811,5.321,148.867
C01395=1227.510,-32.496,-39.571,-179.813,5.322,148.868
C01396=1227.515,-32.746,-39.557,-179.815,5.321,148.869
C01397=1227.520,-32.995,-39.544,-179.818,5.321,148.869
C01398=1227.525,-33.245,-39.531,-179.820,5.321,148.870
C01399=1227.531,-33.495,-39.518,-179.823,5.320,148.871
C01400=1227.536,-33.744,-39.505,-179.825,5.321,148.871
C01401=1227.540,-33.994,-39.492,-179.828,5.320,148.872
C01402=1227.546,-34.244,-39.479,-179.830,5.320,148.873
C01403=1227.551,-34.492,-39.466,-179.832,5.320,148.873
C01404=1227.555,-34.742,-39.453,-179.835,5.320,148.874
C01405=1227.561,-34.992,-39.439,-179.838,5.319,148.875
C01406=1227.566,-35.242,-39.426,-179.840,5.319,148.876
C01407=1227.571,-35.491,-39.414,-179.842,5.319,148.876
C01408=1227.577,-35.741,-39.401,-179.844,5.319,148.877
C01409=1227.581,-35.991,-39.388,-179.847,5.319,148.878
C01410=1227.586,-36.240,-39.375,-179.850,5.318,148.878
C01411=1227.592,-36.490,-39.362,-179.852,5.319,148.879
C01412=1227.597,-36.740,-39.349,-179.855,5.318,148.880
C01413=1227.602,-36.989,-39.336,-179.857,5.318,148.880
C01414=1227.607,-37.238,-39.322,-179.859,5.318,148.881
C01415=1227.612,-37.488,-39.309,-179.862,5.317,148.882
C01416=1227.617,-37.738,-39.297,-179.864,5.318,148.883
C01417=1227.622,-37.987,-39.284,-179.867,5.317,148.883
C01418=1227.628,-38.237,-39.271,-179.869,5.317,148.884
C01419=1227.633,-38.487,-39.258,-179.871,5.317,148.885
C01420=1227.638,-38.736,-39.245,-179.874,5.317,148.885
C01421=1227.642,-38.986,-39.232,-179.876,5.317,148.886
C01422=1227.648,-39.236,-39.219,-179.879,5.317,148.887
C01423=1227.653,-39.485,-39.207,-179.882,5.316,148.888
C01424=1227.658,-39.735,-39.194,-179.884,5.317,148.888
C01425=1227.663,-39.984,-39.181,-179.887,5.316,148.889
C01426=1227.669,-40.234,-39.168,-179.889,5.316,148.890
C01427=1227.673,-40.484,-39.155,-179.892,5.316,148.891
C01428=1227.678,-40.733,-39.142,-179.894,5.315,148.891
C01429=1227.684,-40.983,-39.130,-179.896,5.316,148.892
C01430=1227.688,-41.233,-39.117,-179.899,5.315,148.893
C01431=1227.694,-41.482,-39.104,-179.901,5.316,148.893
C01432=1227.699,-41.732,-39.092,-179.904,5.315,148.894
C01433=1227.704,-41.981,-39.079,-179.906,5.315,148.895
C01434=1227.709,-42.231,-39.066,-179.908,5.315,148.895
C01435=1227.714,-42.481,-39.054,-179.911,5.315,148.896
C01436=1227.719,-42.730,-39.041,-179.913,5.315,148.897
C01437=1227.725,-42.980,-39.027,-179.916,5.314,148.898
C01438=1227.730,-43.230,-39.015,-179.918,5.314,148.898
C01439=1227.735,-43.479,-39.002,-179.921,5.314,148.899
C01440=1227.740,-43.728,-38.990,-179.923,5.314,148.900
C01441=1227.745,-43.979,-38.977,-179.925,5.314,148.900
C01442=1227.750,-44.228,-38.965,-179.928,5.314,148.901
C01443=1227.755,-44.478,-38.952,-179.931,5.313,148.902
C01444=1227.761,-44.727,-38.939,-179.933,5.313,148.902
C01445=1227.765,-44.977,-38.926,-179.935,5.313,148.903
C01446=1227.770,-45.227,-38.913,-179.937,5.313,148.904
C01447=1227.776,-45.477,-38.901,-179.940,5.313,148.905
C01448=1227.781,-45.726,-38.889,-179.943,5.312,148.905
C01449=1227.786,-45.976,-38.876,-179.945,5.313,148.906
C01450=1227.791,-46.225,-38.863,-179.948,5.312,148.907
C01451=1227.796,-46.475,-38.851,-179.950,5.312,148.907
C01452=1227.801,-46.724,-38.839,-179.952,5.312,148.908
C01453=1227.806,-46.974,-38.826,-179.955,5.311,148.909
C01454=1227.812,-47.224,-38.813,-179.957,5.312,148.909
C01455=1227.817,-47.473,-38.800,-179.960,5.311,148.910
C01456=1227.822,-47.723,-38.787,-179.962,5.312,148.911
C01457=1227.827,-47.973,-38.776,-179.964,5.311,148.912
C01458=1227.832,-48.242,-38.762,-179.967,5.311,148.912
C01459=1227.837,-48.512,-38.748,-179.970,5.311,148.913
C01460=1227.844,-48.782,-38.735,-179.972,5.311,148.914
C01461=1227.849,-49.052,-38.721,-179.975,5.310,148.915
C01462=1227.854,-49.301,-38.709,-179.977,5.311,148.915
C01463=1227.859,-49.551,-38.697,-179.980,5.310,148.916
C01464=1227.865,-49.800,-38.684,-179.982,5.311,148.917
C01465=1227.869,-50.050,-38.671,-179.985,5.310,148.917
C01466=1227.875,-50.300,-38.659,-179.987,5.310,148.918
C01467=1227.880,-50.550,-38.647,-179.989,5.310,148.919
C01468=1227.885,-50.799,-38.634,-179.992,5.309,148.920
C01469=1227.890,-51.049,-38.622,-179.994,5.310,148.920
C01470=1227.895,-51.298,-38.610,-179.997,5.309,148.921
C01471=1227.900,-51.548,-38.597,-179.999,5.309,148.922
C01472=1227.905,-51.798,-38.585,179.999,5.309,148.922
C01473=1227.910,-52.048,-38.572,179.996,5.309,148.923
C01474=1227.916,-52.297,-38.560,179.994,5.309,148.924
C01475=1227.921,-52.547,-38.548,179.991,5.308,148.924
C01476=1227.926,-52.796,-38.535,179.989,5.309,148.925
C01477=1227.932,-53.046,-38.523,179.986,5.308,148.926
C01478=1227.936,-53.296,-38.510,179.984,5.308,148.927
C01479=1227.941,-53.545,-38.498,179.981,5.309,148.927
C01480=1227.947,-53.795,-38.486,179.978,5.308,148.928
C01481=1227.951,-54.044,-38.474,179.976,5.308,148.929
C01482=1227.956,-54.294,-38.462,179.974,5.308,148.930
C01483=1227.962,-54.544,-38.449,179.972,5.308,148.930
C01484=1227.967,-54.794,-38.437,179.969,5.308,148.931
C01485=1227.972,-55.043,-38.425,179.966,5.307,148.932
C01486=1227.977,-55.293,-38.412,179.964,5.308,148.932
C01487=1227.982,-55.543,-38.400,179.961,5.307,148.933
C01488=1227.987,-55.792,-38.387,179.959,5.308,148.934
C01489=1227.993,-56.042,-38.375,179.957,5.307,148.935
C01490=1227.998,-56.291,-38.363,179.955,5.307,148.935
C01491=1228.002,-56.541,-38.352,179.952,5.307,148.936
C01492=1228.008,-56.790,-38.339,179.950,5.307,148.937
C01493=1228.013,-57.040,-38.327,179.947,5.307,148.937
C01494=1228.018,-57.290,-38.315,179.945,5.306,148.938
C01495=1228.024,-57.539,-38.303,179.942,5.307,148.939
C01496=1228.029,-57.789,-38.290,179.940,5.306,148.939
C01497=1228.034,-58.039,-38.278,179.938,5.306,148.940
C01498=1228.038,-58.289,-38.266,179.935,5.306,148.941
C01499=1228.043,-58.538,-38.254,179.933,5.306,148.942
C01500=1228.049,-58.788,-38.242,179.930,5.306,148.942
C01501=1228.054,-59.038,-38.229,179.928,5.305,148.943
C01502=1228.059,-59.288,-38.218,179.926,5.306,148.944
C01503=1228.064,-59.537,-38.205,179.923,5.305,148.944
C01504=1228.069,-59.787,-38.194,179.921,5.306,148.945
C01505=1228.075,-60.036,-38.182,179.918,5.305,148.946
C01506=1228.080,-60.286,-38.169,179.916,5.305,148.947
C01507=1228.085,-60.536,-38.157,179.913,5.305,148.947
C01508=1228.089,-60.785,-38.145,179.911,5.305,148.948
C01509=1228.095,-61.035,-38.133,179.909,5.305,148.949
C01510=1228.100,-61.285,-38.121,179.907,5.305,148.949
C01511=1228.105,-61.534,-38.109,179.904,5.305,148.950
C01512=1228.111,-61.784,-38.097,179.901,5.304,148.951
C01513=1228.116,-62.033,-38.086,179.899,5.305,148.951
C01514=1228.121,-62.283,-38.073,179.896,5.304,148.952
C01515=1228.126,-62.533,-38.061,179.894,5.304,148.953
C01516=1228.132,-62.783,-38.049,179.892,5.304,148.954
C01517=1228.136,-63.032,-38.037,179.890,5.304,148.954
C01518=1228.141,-63.282,-38.025,179.887,5.304,148.955
C01519=1228.147,-63.532,-38.014,179.885,5.304,148.956
C01520=1228.152,-63.781,-38.001,179.882,5.304,148.956
C01521=1228.157,-64.030,-37.990,179.879,5.303,148.957
C01522=1228.162,-64.280,-37.978,179.877,5.304,148.958
C01523=1228.167,-64.530,-37.966,179.875,5.303,148.959
C01524=1228.172,-64.779,-37.954,179.873,5.303,148.959
C01525=1228.177,-65.029,-37.942,179.870,5.303,148.960
C01526=1228.183,-65.279,-37.930,179.868,5.303,148.961
C01527=1228.188,-65.529,-37.918,179.865,5.303,148.961
C01528=1228.193,-65.778,-37.906,179.863,5.303,148.962
C01529=1228.198,-66.028,-37.894,179.860,5.303,148.963
C01530=1228.203,-66.278,-37.882,179.858,5.303,148.963
C01531=1228.208,-66.528,-37.871,179.856,5.303,148.964
C01532=1228.213,-66.777,-37.859,179.853,5.302,148.965
C01533=1228.219,-67.027,-37.847,179.851,5.302,148.966
C01534=1228.224,-67.276,-37.836,179.848,5.302,148.966
C01535=1228.229,-67.526,-37.824,179.846,5.302,148.967
C01536=1228.235,-67.776,-37.812,179.844,5.302,148.968
C01537=1228.239,-68.025,-37.801,179.841,5.302,148.968
C01538=1228.245,-68.275,-37.788,179.839,5.302,148.969
C01539=1228.250,-68.525,-37.776,179.837,5.302,148.970
C01540=1228.255,-68.774,-37.765,179.834,5.302,148.971
C01541=1228.260,-69.024,-37.753,179.832,5.302,148.971
C01542=1228.265,-69.274,-37.742,179.829,5.301,148.972
C01543=1228.270,-69.524,-37.730,179.827,5.302,148.973
C01544=1228.276,-69.774,-37.718,179.824,5.301,148.973
C01545=1228.280,-70.023,-37.706,179.822,5.302,148.974
C01546=1228.286,-70.272,-37.694,179.820,5.301,148.975
C01547=1228.291,-70.522,-37.683,179.817,5.301,148.975
C01548=1228.296,-70.771,-37.671,179.815,5.301,148.976
C01549=1228.302,-71.021,-37.659,179.812,5.301,148.977
C01550=1228.306,-71.271,-37.648,179.810,5.301,148.978
C01551=1228.312,-71.521,-37.636,179.808,5.301,148.978
C01552=1228.316,-71.771,-37.625,179.805,5.301,148.979
C01553=1228.322,-72.021,-37.613,179.803,5.300,148.980
C01554=1228.328,-72.270,-37.602,179.801,5.301,148.980
C01555=1228.333,-72.519,-37.590,179.798,5.300,148.981
C01556=1228.338,-72.769,-37.578,179.796,5.301,148.982
C01557=1228.343,-73.019,-37.567,179.793,5.300,148.983
C01558=1228.348,-73.269,-37.555,179.791,5.300,148.983
C01559=1228.353,-73.519,-37.544,179.789,5.300,148.984
C01560=1228.358,-73.768,-37.532,179.786,5.300,148.985
C01561=1228.364,-74.017,-37.521,179.784,5.300,148.985
C01562=1228.369,-74.288,-37.508,179.781,5.299,148.986
C01563=1228.374,-74.558,-37.495,179.779,5.300,148.987
C01564=1228.380,-74.828,-37.483,179.776,5.299,148.988
C01565=1228.386,-75.099,-37.470,179.773,5.299,148.988
C01566=1228.391,-75.349,-37.458,179.771,5.300,148.989
C01567=1228.396,-75.598,-37.447,179.768,5.299,148.990
C01568=1228.402,-75.848,-37.436,179.766,5.299,148.991
C01569=1228.407,-76.097,-37.424,179.764,5.299,148.991
C01570=1228.412,-76.348,-37.413,179.762,5.299,148.992
C01571=1228.417,-76.597,-37.402,179.759,5.299,148.993
C01572=1228.422,-76.847,-37.390,179.757,5.299,148.993
C01573=1228.428,-77.096,-37.379,179.754,5.299,148.994
C01574=1228.432,-77.346,-37.368,179.752,5.299,148.995
C01575=1228.438,-77.596,-37.356,179.749,5.299,148.996
C01576=1228.443,-77.845,-37.345,179.747,5.299,148.996
C01577=1228.448,-78.095,-37.333,179.745,5.299,148.997
C01578=1228.453,-78.344,-37.322,179.742,5.299,148.998
C01579=1228.459,-78.594,-37.310,179.740,5.298,148.998
C01580=1228.464,-78.844,-37.299,179.738,5.298,148.999
C01581=1228.469,-79.094,-37.287,179.736,5.298,149.000
C01582=1228.474,-79.344,-37.276,179.733,5.298,149.000
C01583=1228.479,-79.593,-37.265,179.731,5.298,149.001
C01584=1228.485,-79.843,-37.253,179.729,5.298,149.002
C01585=1228.489,-80.092,-37.242,179.726,5.298,149.002
C01586=1228.495,-80.342,-37.230,179.724,5.298,149.003
C01587=1228.500,-80.592,-37.220,179.721,5.298,149.004
C01588=1228.505,-80.842,-37.209,179.719,5.298,149.005
C01589=1228.510,-81.092,-37.197,179.716,5.298,149.005
C01590=1228.515,-81.341,-37.185,179.714,5.298,149.006
C01591=1228.520,-81.590,-37.175,179.712,5.297,149.007
C01592=1228.526,-81.841,-37.163,179.710,5.298,149.007
C01593=1228.531,-82.090,-37.152,179.707,5.297,149.008
C01594=1228.536,-82.340,-37.140,179.705,5.298,149.009
C01595=1228.542,-82.589,-37.129,179.702,5.297,149.009
C01596=1228.547,-82.839,-37.119,179.700,5.298,149.010
C01597=1228.552,-83.089,-37.107,179.697,5.297,149.011
C01598=1228.557,-83.339,-37.096,179.695,5.297,149.012
C01599=1228.562,-83.588,-37.085,179.693,5.297,149.012
C01600=1228.568,-83.838,-37.073,179.691,5.297,149.013
C01601=1228.572,-84.088,-37.062,179.688,5.297,149.014
C01602=1228.578,-84.337,-37.051,179.686,5.297,149.014
C01603=1228.582,-84.587,-37.040,179.683,5.297,149.015
C01604=1228.588,-84.837,-37.029,179.681,5.297,149.016
C01605=1228.593,-85.087,-37.017,179.678,5.297,149.017
C01606=1228.598,-85.336,-37.007,179.676,5.297,149.017
C01607=1228.604,-85.586,-36.995,179.674,5.297,149.018
C01608=1228.609,-85.836,-36.984,179.672,5.297,149.019
C01609=1228.614,-86.085,-36.973,179.669,5.297,149.019
C01610=1228.619,-86.335,-36.963,179.667,5.297,149.020
C01611=1228.624,-86.585,-36.951,179.664,5.296,149.021
C01612=1228.630,-86.834,-36.940,179.662,5.297,149.022
C01613=1228.635,-87.084,-36.929,179.659,5.296,149.022
C01614=1228.640,-87.334,-36.917,179.657,5.297,149.023
C01615=1228.645,-87.583,-36.906,179.655,5.296,149.024
C01616=1228.650,-87.833,-36.896,179.653,5.296,149.024
C01617=1228.655,-88.083,-36.885,179.650,5.296,149.025
C01618=1228.661,-88.333,-36.874,179.648,5.296,149.026
C01619=1228.666,-88.582,-36.862,179.646,5.296,149.026
C01620=1228.671,-88.832,-36.851,179.643,5.296,149.027
C01621=1228.676,-89.082,-36.841,179.641,5.296,149.028
C01622=1228.681,-89.331,-36.830,179.639,5.296,149.028
C01623=1228.687,-89.582,-36.818,179.636,5.295,149.029
C01624=1228.692,-89.831,-36.808,179.634,5.296,149.030
C01625=1228.697,-90.081,-36.797,179.631,5.295,149.031
C01626=1228.702,-90.330,-36.786,179.629,5.296,149.031
C01627=1228.707,-90.579,-36.775,179.626,5.295,149.032
C01628=1228.713,-90.830,-36.764,179.624,5.296,149.033
C01629=1228.718,-91.079,-36.753,179.622,5.295,149.033
C01630=1228.723,-91.329,-36.742,179.620,5.296,149.034
C01631=1228.728,-91.579,-36.731,179.617,5.295,149.035
C01632=1228.733,-91.828,-36.721,179.615,5.295,149.036
C01633=1228.738,-92.078,-36.709,179.612,5.295,149.036
C01634=1228.744,-92.328,-36.698,179.610,5.295,149.037
C01635=1228.749,-92.577,-36.687,179.607,5.295,149.038
C01636=1228.754,-92.828,-36.677,179.605,5.295,149.038
C01637=1228.759,-93.077,-36.666,179.603,5.295,149.039
C01638=1228.764,-93.327,-36.655,179.601,5.295,149.040
C01639=1228.770,-93.576,-36.644,179.598,5.294,149.040
C01640=1228.775,-93.826,-36.634,179.596,5.295,149.041
C01641=1228.780,-94.077,-36.622,179.594,5.294,149.042
C01642=1228.786,-94.325,-36.612,179.592,5.295,149.042
C01643=1228.791,-94.576,-36.601,179.589,5.294,149.043
C01644=1228.796,-94.825,-36.590,179.587,5.295,149.044
C01645=1228.801,-95.075,-36.579,179.584,5.294,149.045
C01646=1228.806,-95.324,-36.569,179.582,5.294,149.045
C01647=1228.811,-95.574,-36.558,179.579,5.294,149.046
C01648=1228.816,-95.824,-36.547,179.577,5.294,149.047
C01649=1228.821,-96.073,-36.536,179.575,5.294,149.047
C01650=1228.827,-96.324,-36.525,179.572,5.294,149.048
C01651=1228.832,-96.573,-36.514,179.570,5.294,149.049
C01652=1228.837,-96.823,-36.504,179.568,5.294,149.050
C01653=1228.843,-97.072,-36.494,179.565,5.294,149.050
C01654=1228.848,-97.322,-36.482,179.563,5.294,149.051
C01655=1228.853,-97.572,-36.472,179.560,5.294,149.052
C01656=1228.858,-97.822,-36.462,179.558,5.294,149.052
C01657=1228.864,-98.071,-36.451,179.557,5.294,149.053
C01658=1228.869,-98.321,-36.440,179.554,5.294,149.054
C01659=1228.874,-98.571,-36.430,179.552,5.294,149.054
C01660=1228.879,-98.820,-36.419,179.549,5.294,149.055
C01661=1228.885,-99.070,-36.408,179.547,5.294,149.056
C01662=1228.890,-99.320,-36.398,179.544,5.293,149.056
C01663=1228.895,-99.569,-36.387,179.542,5.294,149.057
C01664=1228.900,-99.819,-36.376,179.540,5.293,149.058
C01665=1228.905,-100.069,-36.366,179.537,5.294,149.059
C01666=1228.911,-100.340,-36.354,179.535,5.293,149.059
C01667=1228.916,-100.611,-36.343,179.533,5.294,149.060
C01668=1228.922,-100.882,-36.331,179.530,5.293,149.061
C01669=1228.928,-101.153,-36.320,179.527,5.293,149.062
C01670=1228.933,-101.403,-36.309,179.525,5.294,149.062
C01671=1228.938,-101.652,-36.299,179.523,5.293,149.063
C01672=1228.943,-101.902,-36.288,179.520,5.293,149.064
C01673=1228.949,-102.152,-36.278,179.518,5.293,149.064
C01674=1228.954,-102.402,-36.267,179.516,5.293,149.065
C01675=1228.959,-102.651,-36.257,179.513,5.293,149.066
C01676=1228.964,-102.901,-36.246,179.511,5.293,149.066
C01677=1228.969,-103.151,-36.235,179.509,5.293,149.067
C01678=1228.974,-103.401,-36.225,179.506,5.293,149.068
C01679=1228.980,-103.650,-36.215,179.504,5.293,149.069
C01680=1228.986,-103.900,-36.204,179.501,5.293,149.069
C01681=1228.990,-104.149,-36.193,179.499,5.293,149.070
C01682=1228.996,-104.399,-36.183,179.497,5.293,149.071
C01683=1229.001,-104.649,-36.172,179.495,5.293,149.071
C01684=1229.006,-104.899,-36.162,179.492,5.292,149.072
C01685=1229.011,-105.149,-36.152,179.490,5.293,149.073
C01686=1229.016,-105.398,-36.142,179.488,5.292,149.073
C01687=1229.021,-105.649,-36.131,179.485,5.293,149.074
C01688=1229.027,-105.897,-36.120,179.483,5.292,149.075
C01689=1229.032,-106.147,-36.110,179.481,5.292,149.076
C01690=1229.037,-106.397,-36.100,179.478,5.292,149.076
C01691=1229.043,-106.647,-36.089,179.476,5.292,149.077
C01692=1229.048,-106.897,-36.079,179.473,5.292,149.078
C01693=1229.053,-107.146,-36.069,179.471,5.292,149.078
C01694=1229.058,-107.396,-36.059,179.469,5.293,149.079
C01695=1229.063,-107.646,-36.049,179.466,5.292,149.080
C01696=1229.069,-107.896,-36.038,179.465,5.292,149.080
C01697=1229.074,-108.146,-36.028,179.462,5.292,149.081
C01698=1229.079,-108.395,-36.018,179.460,5.292,149.082
C01699=1229.085,-108.644,-36.007,179.457,5.292,149.082
C01700=1229.089,-108.894,-35.997,179.455,5.292,149.083
C01701=1229.095,-109.144,-35.986,179.453,5.292,149.084
C01702=1229.100,-109.394,-35.976,179.451,5.292,149.085
C01703=1229.105,-109.644,-35.966,179.448,5.292,149.085
C01704=1229.111,-109.893,-35.955,179.446,5.292,149.086
C01705=1229.116,-110.143,-35.945,179.443,5.292,149.087
C01706=1229.121,-110.393,-35.935,179.441,5.292,149.087
C01707=1229.126,-110.642,-35.925,179.439,5.292,149.088
C01708=1229.131,-110.892,-35.914,179.437,5.291,149.089
C01709=1229.137,-111.142,-35.904,179.435,5.292,149.089
C01710=1229.142,-111.391,-35.894,179.432,5.291,149.090
C01711=1229.147,-111.641,-35.884,179.430,5.292,149.091
C01712=1229.152,-111.891,-35.874,179.427,5.291,149.092
C01713=1229.158,-112.140,-35.864,179.425,5.292,149.092
C01714=1229.163,-112.391,-35.854,179.422,5.291,149.093
C01715=1229.168,-112.641,-35.844,179.420,5.292,149.094
C01716=1229.174,-112.890,-35.834,179.418,5.291,149.094
C01717=1229.179,-113.140,-35.823,179.416,5.291,149.095
C01718=1229.184,-113.390,-35.813,179.413,5.291,149.096
C01719=1229.189,-113.639,-35.804,179.411,5.291,149.096
C01720=1229.194,-113.889,-35.793,179.409,5.292,149.097
C01721=1229.200,-114.139,-35.783,179.406,5.291,149.098
C01722=1229.205,-114.388,-35.773,179.404,5.291,149.098
C01723=1229.210,-114.638,-35.763,179.402,5.291,149.099
C01724=1229.215,-114.888,-35.752,179.400,5.291,149.100
C01725=1229.221,-115.137,-35.742,179.397,5.291,149.100
C01726=1229.225,-115.388,-35.733,179.395,5.291,149.101
C01727=1229.231,-115.638,-35.723,179.393,5.291,149.102
C01728=1229.237,-115.887,-35.712,179.391,5.291,149.102
C01729=1229.242,-116.137,-35.702,179.388,5.291,149.103
C01730=1229.246,-116.387,-35.692,179.386,5.291,149.104
C01731=1229.252,-116.636,-35.682,179.384,5.291,149.105
C01732=1229.258,-116.886,-35.673,179.381,5.291,149.105
C01733=1229.262,-117.136,-35.663,179.379,5.291,149.106
C01734=1229.268,-117.386,-35.652,179.377,5.290,149.107
C01735=1229.273,-117.635,-35.642,179.375,5.291,149.107
C01736=1229.278,-117.885,-35.633,179.372,5.290,149.108
C01737=1229.283,-118.135,-35.622,179.370,5.291,149.109
C01738=1229.289,-118.385,-35.613,179.367,5.290,149.109
C01739=1229.294,-118.634,-35.603,179.365,5.291,149.110
C01740=1229.300,-118.884,-35.593,179.362,5.290,149.111
C01741=1229.305,-119.134,-35.582,179.361,5.290,149.111
C01742=1229.310,-119.384,-35.573,179.359,5.291,149.112
C01743=1229.315,-119.633,-35.563,179.356,5.290,149.113
C01744=1229.320,-119.883,-35.553,179.354,5.291,149.113
C01745=1229.325,-120.133,-35.543,179.351,5.290,149.114
C01746=1229.331,-120.383,-35.533,179.349,5.291,149.115
C01747=1229.336,-120.632,-35.524,179.346,5.290,149.116
C01748=1229.342,-120.882,-35.514,179.345,5.290,149.116
C01749=1229.346,-121.132,-35.504,179.342,5.290,149.117
C01750=1229.352,-121.382,-35.494,179.340,5.290,149.118
C01751=1229.357,-121.631,-35.484,179.338,5.290,149.118
C01752=1229.362,-121.881,-35.474,179.335,5.290,149.119
C01753=1229.368,-122.132,-35.464,179.333,5.290,149.120
C01754=1229.372,-122.381,-35.455,179.331,5.290,149.120
C01755=1229.378,-122.630,-35.445,179.329,5.290,149.121
C01756=1229.383,-122.880,-35.436,179.326,5.290,149.122
C01757=1229.389,-123.130,-35.425,179.324,5.290,149.122
C01758=1229.394,-123.380,-35.415,179.321,5.289,149.123
C01759=1229.399,-123.630,-35.406,179.319,5.290,149.124
C01760=1229.404,-123.879,-35.396,179.317,5.290,149.124
C01761=1229.409,-124.129,-35.386,179.315,5.290,149.125
C01762=1229.415,-124.379,-35.377,179.313,5.290,149.126
C01763=1229.420,-124.628,-35.367,179.310,5.289,149.126
C01764=1229.425,-124.878,-35.356,179.308,5.290,149.127
C01765=1229.430,-125.128,-35.348,179.306,5.289,149.128
C01766=1229.436,-125.378,-35.337,179.303,5.290,149.129
C01767=1229.441,-125.627,-35.328,179.301,5.289,149.129
C01768=1229.447,-125.877,-35.318,179.299,5.290,149.130
C01769=1229.451,-126.127,-35.308,179.297,5.290,149.130
C01770=1229.030,-126.138,-35.344,179.292,5.292,149.133
C01771=1229.025,-125.888,-35.355,179.295,5.293,149.132
C01772=1229.020,-125.638,-35.364,179.297,5.292,149.131
C01773=1229.014,-125.388,-35.374,179.299,5.293,149.130
C01774=1229.009,-125.138,-35.383,179.301,5.293,149.130
C01775=1229.003,-124.889,-35.393,179.304,5.293,149.129
C01776=1228.998,-124.640,-35.402,179.306,5.293,149.129
C01777=1228.993,-124.389,-35.412,179.309,5.293,149.128
C01778=1228.988,-124.140,-35.422,179.311,5.293,149.127
C01779=1228.982,-123.889,-35.431,179.313,5.293,149.126
C01780=1228.978,-123.640,-35.441,179.315,5.293,149.126
C01781=1228.972,-123.391,-35.451,179.317,5.293,149.125
C01782=1228.966,-123.141,-35.461,179.320,5.293,149.124
C01783=1228.962,-122.891,-35.471,179.322,5.293,149.124
C01784=1228.956,-122.641,-35.481,179.324,5.293,149.123
C01785=1228.951,-122.391,-35.490,179.327,5.293,149.122
C01786=1228.945,-122.142,-35.500,179.329,5.294,149.122
C01787=1228.941,-121.892,-35.510,179.331,5.294,149.121
C01788=1228.935,-121.642,-35.519,179.333,5.293,149.120
C01789=1228.930,-121.392,-35.530,179.336,5.294,149.120
C01790=1228.925,-121.143,-35.539,179.338,5.293,149.119
C01791=1228.919,-120.893,-35.550,179.340,5.294,149.118
C01792=1228.915,-120.643,-35.559,179.342,5.293,149.118
C01793=1228.909,-120.393,-35.569,179.345,5.294,149.117
C01794=1228.904,-120.144,-35.579,179.347,5.294,149.116
C01795=1228.898,-119.894,-35.588,179.349,5.294,149.116
C01796=1228.893,-119.643,-35.599,179.352,5.294,149.115
C01797=1228.888,-119.394,-35.608,179.354,5.294,149.114
C01798=1228.883,-119.145,-35.618,179.356,5.294,149.113
C01799=1228.877,-118.895,-35.628,179.358,5.293,149.113
C01800=1228.873,-118.645,-35.638,179.361,5.294,149.112
C01801=1228.867,-118.395,-35.648,179.363,5.294,149.112
C01802=1228.861,-118.146,-35.658,179.365,5.294,149.111
C01803=1228.857,-117.896,-35.668,179.367,5.294,149.110
C01804=1228.851,-117.645,-35.678,179.370,5.294,149.109
C01805=1228.846,-117.396,-35.687,179.372,5.294,149.109
C01806=1228.841,-117.147,-35.698,179.375,5.294,149.108
C01807=1228.835,-116.897,-35.708,179.377,5.294,149.107
C01808=1228.831,-116.647,-35.718,179.379,5.294,149.107
C01809=1228.825,-116.398,-35.728,179.381,5.294,149.106
C01810=1228.819,-116.147,-35.738,179.383,5.294,149.105
C01811=1228.814,-115.897,-35.748,179.386,5.294,149.105
C01812=1228.810,-115.648,-35.758,179.388,5.294,149.104
C01813=1228.804,-115.398,-35.768,179.391,5.295,149.103
C01814=1228.798,-115.149,-35.778,179.393,5.294,149.102
C01815=1228.794,-114.899,-35.788,179.396,5.295,149.102
C01816=1228.789,-114.649,-35.798,179.398,5.294,149.101
C01817=1228.783,-114.399,-35.808,179.400,5.295,149.100
C01818=1228.778,-114.149,-35.818,179.402,5.295,149.100
C01819=1228.773,-113.900,-35.828,179.405,5.295,149.099
C01820=1228.767,-113.650,-35.838,179.407,5.295,149.098
C01821=1228.762,-113.400,-35.849,179.409,5.294,149.098
